(* CoDeSys 2.3.9.59 project: Festo_Project_Group_S.pro *)
(* Title: Tesi *)
(* Version: Studenti *)
(* Author: Marco Pierantoni *)
(* Libraries: STANDARD.LIB 4.10.05 11:14:46, IECSFC.LIB 2.6.14 10:37:46, ANALYZATION.LIB 2.6.14 10:37:46 *)

(* Task configuration *)
TASK SimulationTask (PRIORITY := 1, INTERVAL := T#1ms);
	Pulsantiera();
	PlantCarico();
	PlantScarico();
	PlantMagazzino();
	PlantVerification();
	PlantLavorazione();
	PlantAssemblaggio();
END_TASK
TASK Main (PRIORITY := 1, INTERVAL := T#2ms);
	InputBridge();
	Main();
	OutputBridge();
END_TASK

(* Global variable list: SignalManagement/FaultVariables_List *)
VAR_GLOBAL
(*FAULT VAR*) (* Used as ActivationSignal for SignalManagment *)

	(* Station ONE *)

	F_Cylinder1: BOOL;
	F_S_Cylinder1: BOOL;
	F_A_Cylinder1: BOOL;
	FH_A_Cylinder1: BOOL;
	FL_A_Cylinder1: BOOL;
	FL_DS_Cylinder1: BOOL;
	FH_DS_Cylinder1: BOOL;
	FL_ES_Cylinder1: BOOL;
	FH_ES_Cylinder1: BOOL;

	F_Rotary1: BOOL;
	F_S_Rotary1: BOOL;
	F_A_Rotary1 : BOOL;
	FL_EA_Rotary1: BOOL;
	FH_EA_Rotary1: BOOL;
	FL_DA_Rotary1: BOOL;
	FH_DA_Rotary1: BOOL;
	FL_ES_Rotary1: BOOL;
	FH_ES_Rotary1: BOOL;
	FL_DS_Rotary1: BOOL;
	FH_DS_Rotary1: BOOL;

	F_Vacuum1: BOOL;
	F_S_Vacuum1: BOOL;
	F_A_Vacuum1: BOOL;
	FH_A_Vacuum1: BOOL;
	FL_A_Vacuum1: BOOL;
	FH_S_Vacuum1: BOOL;
	FL_S_Vacuum1: BOOL;

	F_Expulsion1: BOOL;				(* THINK DIAGNOSTIC *)
	F_A_Expulsion1 : BOOL;
	FH_A_Expulsion1: BOOL;
	FL_A_Expulsion1: BOOL;

	(* Station TWO *)

	F_Elevator2: BOOL;
	F_S_Elevator2: BOOL;
	F_A_Elevator2: BOOL;
	FH_EA_Elevator2: BOOL;
	FL_EA_Elevator2: BOOL;
	FH_DA_Elevator2: BOOL;
	FL_DA_Elevator2: BOOL;
	FH_ES_Elevator2: BOOL;
	FL_ES_Elevator2: BOOL;
	FH_DS_Elevator2: BOOL;
	FL_DS_Elevator2: BOOL;

	F_Cylinder2: BOOL;
	F_S_Cylinder2: BOOL;
	F_A_Cylinder2: BOOL;
	FH_A_Cylinder2 : BOOL;
	FL_A_Cylinder2 : BOOL;
	FH_S_Cylinder2 : BOOL;
	FL_S_Cylinder2 : BOOL;

	F_Air2: BOOL;				(* THINK DIAGNOSTIC *)
	F_S_Air2: BOOL;
	F_A_Air2: BOOL;
	FH_A_Air2: BOOL;
	FL_A_Air2: BOOL;

	(* Station THREE *)

	F_RotaryTable3: BOOL;
	F_S_RotaryTable3: BOOL;
	F_A_RotaryTable3: BOOL;
	FH_A_RotaryTable3: BOOL;
	FL_A_RotaryTable3: BOOL;
	FH_S_RotaryTable3: BOOL;
	FL_S_RotaryTable3: BOOL;

	F_Cylinder3: BOOL;		(* THINK DIAGNOSTIC *)
	F_S_Cylinder3: BOOL;
	F_A_Cylinder3: BOOL;
	FH_A_Cylinder3: BOOL;
	FL_A_Cylinder3: BOOL;

	F_DrillCylinder3: BOOL;
	F_S_DrillCylinder3: BOOL;
	F_A_DrillCylinder3: BOOL;
	FH_EA_DrillCylinder3: BOOL;
	FL_EA_DrillCylinder3: BOOL;
	FH_DA_DrillCylinder3: BOOL;
	FL_DA_DrillCylinder3: BOOL;
	FH_ES_DrillCylinder3: BOOL;
	FL_ES_DrillCylinder3: BOOL;
	FH_DS_DrillCylinder3: BOOL;
	FL_DS_DrillCylinder3: BOOL;

	F_Drilling3: BOOL;			(* THINK DIAGNOSTIC *)
	F_S_Drilling3: BOOL;
	F_A_Drilling3: BOOL;
	FH_A_Drilling3: BOOL;
	FL_A_Drilling3: BOOL;

	F_Block3: BOOL;			(* THINK DIAGNOSTIC *)
	F_S_Block3: BOOL;
	F_A_Block3: BOOL;
	FH_A_Block3: BOOL;
	FL_A_Block3: BOOL;

	F_Expell3: BOOL;				(* THINK DIAGNOSTIC *)
	F_S_Expell3: BOOL;
	F_A_Expell3: BOOL;
	FH_A_Expell3: BOOL;
	FL_A_Expell3: BOOL;

	(* Station FOUR *)

	F_SpringExtractor4: BOOL;
	F_S_SpringExtractor4: BOOL;
	F_A_SpringExtractor4: BOOL;
	FH_A_SpringExtractor4: BOOL;
	FL_A_SpringExtractor4: BOOL;
	FH_ES_SpringExtractor4: BOOL;
	FL_ES_SpringExtractor4: BOOL;
	FH_DS_SpringExtractor4: BOOL;
	FL_DS_SpringExtractor4: BOOL;

	F_PistonSelector4: BOOL;
	F_S_PistonSelector4: BOOL;
	F_A_PistonSelector4: BOOL;
	FH_EA_PistonSelector4: BOOL;
	FL_EA_PistonSelector4: BOOL;
	FH_DA_PistonSelector4: BOOL;
	FL_DA_PistonSelector4: BOOL;
	FH_ES_PistonSelector4: BOOL;
	FL_ES_PistonSelector4: BOOL;
	FH_DS_PistonSelector4: BOOL;
	FL_DS_PistonSelector4: BOOL;

	F_ExtractCover4: BOOL;
	F_S_ExtractCover4: BOOL;
	F_A_ExtractCover4: BOOL;
	FH_A_ExtractCover4: BOOL;
	FL_A_ExtractCover4: BOOL;
	FH_ES_ExtractCover4: BOOL;
	FL_ES_ExtractCover4: BOOL;
	FH_DS_ExtractCover4: BOOL;
	FL_DS_ExtractCover4: BOOL;

	F_BlockingCylinder4: BOOL;		(* THINK DIAGNOSTIC *)
	F_S_BlockingCylinder4: BOOL;
	F_A_BlockingCylinder4: BOOL;
	FH_A_BlockingCylinder4: BOOL;
	FL_A_BlockingCylinder4: BOOL;

	(* Robot Manipulator *)

	F_A_RobotToInitial4: BOOL;
	F_S_RobotInInitial4: BOOL;
	(*F_A_RobotTakeBlack4: BOOL;
	F_A_RobotTakeRedSilver4: BOOL;
	F_A_RobotDiscardBlack4: BOOL;
	F_A_RobotDiscardRedSilver4: BOOL;*)
	F_A_RobotAssembly4: BOOL;
	F_S_RobotAssembly4: BOOL;
	F_A_RobotPiston4: BOOL;
	F_S_RobotPiston4: BOOL;
	F_A_RobotSpring4: BOOL;
	F_S_RobotSpring4: BOOL;
	F_A_RobotCover4: BOOL;
	F_S_RobotCover4: BOOL;
	(*F_A_RobotReset4: BOOL;*)

END_VAR

(* Global variable list: MyGlobal/GenericDeviceLib *)
(*Feedback*)

VAR_GLOBAL CONSTANT
	DEVICE_WITHOUT_FEEDBACK : BYTE := 2#01000000;
	DEVICE_WITH_ENABLE_FEEDBACK : BYTE := 2#00010000;
	DEVICE_WITH_DISABLE_FEEDBACK : BYTE := 2#00100000;
	DEVICE_WITH_DOUBLE_FEEDBACK : BYTE := 2#00110000;
	DEVICE_FEEDBACK_MASK : BYTE := 2#11110000;
END_VAR

(*Actuation*)

VAR_GLOBAL CONSTANT
	DEVICE_WITH_SINGLE_ACTUATION : BYTE := 2#00000001;
	DEVICE_WITH_DOUBLE_ACTUATION : BYTE := 2#00000011;
	DEVICE_WITH_DA_NO_RETAIN : BYTE := 2#00000010;
	DEVICE_ACTUATION_MASK : BYTE := 2#00001111;
END_VAR

(* Global variable list: MyGlobal/My_global *)
VAR_GLOBAL CONSTANT

	INIT : INT := 1;
	RUN : INT := 2;
	IMMEDIATESTOPMACHINE : INT :=3;
	READYTORESET : INT:= 4;
	READYTORUN : INT := 5;
	ONPHASESTOPMACHINE : INT := 6;
	EMERGENCYSTOPMACHINE : INT := 7;

END_VAR

VAR_GLOBAL

	BridgeInitOperation : BOOL := TRUE; (* USED ONLY for RealPlant *)
	SignHandlerOperationType : INT ;
	DeviceClock : BOOL;
	OperationType : INT;
	KeyReset : BOOL;
	CumulativeReset : BOOL;
	NoSignalsToReset : BOOL;
	OUTPUT_COUNTER_DELAY : INT := 5; (* Used for Provisional Reset , equal for all by design*)
	SensorActuationDiagnosticEnabled : BOOL := TRUE;

	AllStationsIdle: BOOL; (*Needed For Auto-Stop in case of Inactivity*)

	EmergencyInStop : BOOL;
	ImmediateInStop : BOOL;
	OnPhaseInStop : BOOL;

	(* Necessary on Virtual Panel *)

	VL_StateInit: BOOL;
	VL_StateReady: BOOL;
	VL_StateRun: BOOL;
	VL_StateAlarm: BOOL;
	VL_StateImmediateStop: BOOL;
	VL_StateStop: BOOL;
	VL_StateReset: BOOL;

	VL_ColorVis2:DWORD;
	VL_ColorVis3:DWORD;
	VL_ColorVis:DWORD;
	VL_PositionVis: DWORD;
	VL_ColorVis4:DWORD;
	VL_Completed: INT;
	VL_Rejected: INT;

	(* Used for Station 4 *)

	SpringHouseNotEmpty: BOOL;
	B_SpringLoader: BOOL;
	NumSpring: INT := 0;
	B_PistonLoader: BOOL;
	PistonHouseNotEmpty: BOOL;
	NumPistonBlack: INT;
	NumPistonGrey: INT;

	(*Needed global for real plant for filters*)
	(*Clock2ms: BOOL;
	Clock10ms: BOOL;
	Clock100ms: BOOL;
	Clock1s: BOOL;*)

END_VAR

(* Global variable list: MyGlobal/MyBridgedVariables *)
VAR_GLOBAL

(******* My Variables for Sensors (S), Actuators (A), Lights (L) and Buttons (B)  ***************)

	(* Distribution Station *)

	S_EmptyWarehouse1: BOOL;
	S_CylinderExtended1:BOOL;
	A_Cylinder1: BOOL;
	S_CylinderRetracted1: BOOL;
	A_ArmToWarehouse1: BOOL;
	A_ArmToElevator1: BOOL;
	S_ArmInWarehouse1: BOOL;
	S_ArmInElevator1: BOOL;
	A_Vacuum1: BOOL;
	S_VacuumOk1: BOOL;
	A_AirVacuum1: BOOL;

	(* Verification/Testing Station *)

	S_InterferenceArmElevator2: BOOL;
	A_ElevatorUp2: BOOL;
	A_ElevatorDown2: BOOL;
	S_IsElevatorUp2: BOOL;
	S_IsElevatorDown2: BOOL;
	A_Cylinder2: BOOL;
	S_CylinderExtended2: BOOL;
	S_CylinderRetracted2: BOOL;
	A_AirSlider2: BOOL;
	S_ElementInElevator2: BOOL;
	S_Color2: BOOL;
	S_IsHigh2: BOOL;

	(* Processing Station *)

	A_RotaryTable3: BOOL;
	S_RotaryAlligned3: BOOL;
	S_AvaiableElement3: BOOL;
	S_ControlElement3: BOOL;
	S_DrillElement3: BOOL;
	A_GoControl3: BOOL;
	S_IsOnTheRightSide3: BOOL;
	A_GoDrill3: BOOL;
	A_ReturnDrill3: BOOL;
	S_DrillUp3: BOOL;
	S_DrillDown3: BOOL;
	A_Drilling3: BOOL;
	A_BlockElement3: BOOL;
	A_ExpellElement3: BOOL;

	(* Assembly Station *)

	A_SpringCylinder4: BOOL;
	S_SpringCylinderExtended4: BOOL;
	S_SpringCylinderRetracted4: BOOL;
	A_GiveBlackPiston4: BOOL;
	A_GiveSilverPiston4: BOOL;
	S_BlackPistonGiven4: BOOL;
	S_SilverPistonGiven4: BOOL;
	A_CoverCylinder4: BOOL;
	S_NoCover4: BOOL;
	S_CoverCylinderRetracted4: BOOL;
	S_CoverCylinderExtracted4: BOOL;
	S_ElementAvailable4: BOOL;
	A_BlockElement4: BOOL;

	(* Robot Manipulator *)

	A_RobotToInitial4: BOOL;
	S_RobotInInitial4: BOOL;
	A_RobotTakeBlack4: BOOL;
	A_RobotTakeRedSilver4: BOOL;
	A_RobotDiscardBlack4: BOOL;
	 A_RobotDiscardRedSilver4: BOOL;
	A_RobotAssembly4: BOOL;
	S_RobotAssembly4: BOOL;
	A_RobotPiston4: BOOL;
	S_RobotPiston4: BOOL;
	A_RobotSpring4: BOOL;
	S_RobotSpring4: BOOL;
	A_RobotCover4: BOOL;
	S_RobotCover4: BOOL;
	A_RobotReset4: BOOL;
	StopOutput4 : BOOL := FALSE;

	(* Buttons and Lights *)

	B_Start: BOOL;
	L_Start: BOOL;
	B_Reset: BOOL;
	L_Reset: BOOL;
	B_Stop: BOOL;
	B_Freeze: BOOL;
	B_Emergency: BOOL;
	L_PieceToDiscard2 : BOOL;
	L_EmptyWarehouse: BOOL;
	B_FullWarehouse: BOOL;
	L_UpsideDownElement: BOOL;
	L_NoCover: BOOL;
	B_OnlyBlackElement: BOOL;
	B_AllColors: BOOL;
	B_FaultyElementRemoved: BOOL;
	L_RobotMoving: BOOL;
	L_RobotOn: BOOL;
	L_BlackElement: BOOL;
	L_RedSilverElement: BOOL;
	B_FillAll:BOOL;

END_VAR

(* Global variable list: SignalManagement/SignalCodes_List *)
VAR_GLOBAL

	(*FAULT MESSAGE*) (* "SignalCodes" *)

	(* ALARMS : 1-70 *)

	(*ANOMALIES : 71-130 *)

	(* Warnings: 131 - 190 *)

	(* Informations : 191 - 256 *)

(************************************************************************************************************************************)

	(* Each type has first 10 for Others, 10 for S1, 10 for S2, 10 for S3, 10 for S4 and 10 or more for Others *)

	(*PRIORITARY ALARMS *)

	mEmergencyButtonPressed : WORD := 0003;
	mFreezeButtonPressed : WORD := 0004;
	mOnPhaseStopButtonPressed : WORD := 0005;

	(* WARNINGS *)

	mIdleStopAutoRequest : WORD := 00131;

	(* INFORMATIONS *)

	mEmptyWarehouse : WORD := 00191;
	mEmpyCoverInAssembly : WORD := 00198;

	(*DISTRIBUTION STATION *)

	mS1CylinderActuationFault : WORD := 00021;				mS1CylinderSensorFault : WORD := 00081;
	mS1ArmActuationFault : WORD := 00023;					mS1ArmSensorFault : WORD := 00084;
	mS1VacuumActuationFault : WORD := 00026; 				mS1VacuumSensorFault : WORD := 00087;
	mS1ExpulsionAirActuationFault : WORD := 00028;

	(*VERIFICATION STATION *)

	mS2ElevatorActuationFault : WORD := 00031; 		 		mS2ElevatorSensorFault : WORD := 00091;
	mS2CylinderActuationFault : WORD := 00034; 		 		mS2CylinderSensorFault : WORD := 00094;
	mS2AirSliderActuationFault : WORD := 00036;
	
	(*PROCESSING STATION *)

	mS3RotaryActuationFault : WORD := 00041;	 		  		mS3RotarySensorFault : WORD := 00101;
	mS3InspectorActuationFault : WORD := 00043;	
	mS3DrillCylinderActuationFault : WORD := 00045; 	  		mS3DrillCylinderSensorFault : WORD := 00103;
	mS3DrilerActuationFault : WORD := 00047;
	mS3BlockerActuationFault : WORD := 00048;
	mS3ExpellerActuationFault : WORD := 00049;

	(*ASSEMBLY STATION *)

	mS4SpringExtractorActuationFault : WORD := 00051;		mS4SpringExtractorSensorFault : WORD := 00111;
	mS4PistonSelectorActuationFault : WORD := 00052;		mS4PistonSelectorSensorFault : WORD := 00112;
	mS4CoverExtractorActuationFault : WORD := 00053;		mS4CoverExtractorSensorFault: WORD := 00113;
	mS4BlockerActuationFault : WORD := 00054;

	(* ROBOT MANIPULATOR *)

	mS4RobotInitActuationFault : WORD := 00056;				mS4RobotInitSensorFault : WORD := 00115;
	mS4RobotPistonActuationFault : WORD := 00057;			mS4RobotPistonSensorFault : WORD := 00116;
	mS4RobotSpringActuationFault : WORD := 00058;			mS4RobotSpringSensorFault : WORD := 00117;
	mS4RobotCoverActuationFault : WORD := 00059;			mS4RobotCoverSensorFault : WORD := 00118;
	mS4RobotAssemblyActuationFault : WORD := 00060;		mS4RobotAssemblySensorFault : WORD := 00119;

END_VAR

(* Global variable list: SignalManagement/SignalConstants *)
VAR_GLOBAL CONSTANT
(* OperationTypes *)

(*	INIT : INT :=1;	*)

	START_CONFIGURATION : INT := 12;
	CONFIGURATION : INT := 13;
	START_GENERATION : INT := 14;
	GENERATION : INT := 15;

(* SignalTypes *)

	ALARM : WORD := 00001;
	ANOMALY : WORD := 00002;
	WARNING : WORD := 00003;
	INFORMATION : WORD := 00004;
	SIGNAL_TYPE_MASK : WORD := 00007;

(* ResetTypes *)

	AUX_RESET : WORD := 512;			 (* Reset enabled only if aux reset input active *)
	AUTO_RESET : WORD := 1024;		(* IF ActivationSignal is not present anymore *)
	AUTO_CONDITIONED_RESET : WORD := 2048;	(* IF ActivatSignal not pres anymore AND IF AutoResetSignal TRUE *)
	UNCONDITIONED_RESET : WORD := 4096;		(* Reset in any case if most important *)

	AUTO_PROVISIONAL_RESET : WORD := 8192;
	AUTO_PRIORITY_RESET : WORD := 16384;

(* SignalOutputs *)

	NONE : DWORD := 16#000;

	EMERGENCY_STOP : DWORD := 16#0001;
	IMMEDIATE_STOP : DWORD := 16#0002;
	ON_PHASE_STOP : DWORD := 16#0004;

END_VAR

(* Global variable list: SIM_Global_Variables *)
VAR_GLOBAL


(*------------------------------------------------------------------------------------------------------------------------------------------------*)
(*-----------------------------------VARIABILI DI VISUALIZZAZIONE DEGLI ELEMENTI----------------------------------------*)

(********************variabili utilizzate solo per la simulazione (NON per la logica di controllo)**********************)

(*---------Elementi presenti nel magazzino basi: il magazzino può contenere al più 8 elementi---------*)
	ElementOneCharged: BOOL; (*variabile che indica la presenza del primo elemento nel magazzino*)
	ElementTwoCharged: BOOL; (*secondo elemento caricato nel magazzino*)
	ElementThreeCharged: BOOL; (*terzo elemento caricato nel magazzino*)
	ElementFourCharged: BOOL; (*quarto elemento caricato nel magazzino*)
	ElementFiveCharged: BOOL; (*quinto elemento caricato nel magazzino*)
	ElementSixCharged: BOOL; (*sesto elemento caricato nel magazzino*)
	ElementSevenCharged: BOOL; (*settimo elemento caricato nel magazzino*)
	ElementEightCharged: BOOL; (*ottavo e ultimo elemento caricato nel magazzino*)

(*colori. I possibili colori degli elementi caricabili sono: Rosso, Nero e Argentato (o Metallico)*)
	Red: BOOL; (*è stato caricato un pezzo rosso*)
	Black: BOOL; (*è stato caricato un pezzo nero*)
	Silver: BOOL; (*è stato caricato un pezzo argentato*)

(*pezzi rossi*)
	ElementOneRed: BOOL; (*variabile che indica che il primo elemento caricato è rosso*)
	ElementTwoRed: BOOL; (*il secondo elemento caricato è rosso*)
	ElementThreeRed: BOOL; (*il terzo elemento caricato è rosso*)
	ElementFourRed: BOOL; (*il quarto elemento caricato è rosso*)
	ElementFiveRed: BOOL; (*il quinto elemento caricato è rosso*)
	ElementSixRed: BOOL; (*il sesto elemento caricato è rosso*)
	ElementSevenRed: BOOL; (*il settimo elemento caricato è rosso*)
	ElementEightRed: BOOL; (*l'ottavo elemento caricato è rosso*)

 (*pezzi metallici*)
	ElementOneSilver: BOOL; (*variabile che indica che il primo elemento caricato è argentato*)
	ElementTwoSilver: BOOL;
	ElementThreeSilver: BOOL;
	ElementFourSilver: BOOL;
	ElementFiveSilver: BOOL;
	ElementSixSilver: BOOL;
	ElementSevenSilver: BOOL;
	ElementEightSilver: BOOL;

 (*pezzi neri*)
	ElementOneBlack: BOOL; (*variabile che indica che il primo elemento caricato è nero*)
	ElementTwoBlack: BOOL;
	ElementThreeBlack: BOOL;
	ElementFourBlack: BOOL;
	ElementFiveBlack: BOOL;
	ElementSixBlack: BOOL;
	ElementSevenBlack: BOOL;
	ElementEightBlack: BOOL;

(*-----pezzi capovolti-----Può capitare che alcune basi vengano caricate capovolte nel magazzino: le variabili seguenti simulano questa ipotesi*)
	Redoverturned: BOOL; (*variabile che indica che l'elemento rosso è capovolto*)
	Silveroverturned: BOOL; (*variabile che indica che l'elemento argentato è capovolto*)
	Blackoverturned: BOOL; (*variabile che indica che l'elemento nero è capovolto*)

(*---------Elementi caricati capovolti nel magazzino basi--------*)
	ElementOneOverturned: BOOL; (*variabile che indica che il primo elemento del magazzino è stato caricato capovolto*)
	ElementTwoOverturned: BOOL; (*secondo elemento del magazzino caricato capovolto*)
	ElementThreeOverturned: BOOL; (*terzo elemento del magazzino caricato capovolto*)
	ElementFourOverturned: BOOL; (*quarto elemento del magazzino caricato capovolto*)
	ElementFiveOverturned: BOOL; (*quinto elemento del magazzino caricato capovolto*)
	ElementSixOverturned: BOOL; (*sesto elemento del magazzino caricato capovolto*)
	ElementSevenOverturned: BOOL; (*settimo elemento del magazzino caricato capovolto*)
	ElementEightOverturned: BOOL; (*ottavo elemento del magazzino caricato capovolto*)

(*----pezzi corti:
I pezzi chiari (rossi/met) sono alti, quelli neri, bassi. Può capitare che nel magazzino vengano caricati pezzi chiari ma bassi per difetti di costruzione:
le variabili seguenti simulano questa ipotesi*)

(*per la simulazione è stato creato solo il pezzo metallico corto: non è necessario creare anche quello rosso perchè il sistema non distingue tra rosso e metallico ma solo tra chiaro e nero*)
	Silvershort: BOOL; (*pezzo argentato corto*)

(*---------Elementi corti caricati nel magazzino basi--------*)
	ElementOneShort: BOOL; (*il primo elemento del magazzino è corto*)
	ElementTwoShort: BOOL;
	ElementThreeShort: BOOL;
	ElementFourShort: BOOL;
	ElementFiveShort: BOOL;
	ElementSixShort: BOOL;
	ElementSevenShort: BOOL;
	ElementEightShort: BOOL;

(*stringhe di segnalazione pezzo capovolto o corto: viene visualizzata una O se il pezzo è capovolto oppure una S se è corto. Niente altrimenti.*)
	ElementOneO: STRING; (*sul primo elemento del magazzino viene visualizzata stringa "O"(Overturned), oppure "S" (Short), oppure "" (pezzo normale)*)
	ElementTwoO: STRING;
	ElementThreeO: STRING;
	ElementFourO: STRING;
	ElementFiveO: STRING;
	ElementSixO: STRING;
	ElementSevenO: STRING;
	ElementEightO: STRING;

(*-----Elemento in Attesa: una volta espulso dal magazzino basi l'elemento rimane in attesa di essere caricato dal braccio rotante-----*)
	ElementWaitingCharged: BOOL; (*variabile che indica che è presente un elemento in attesa*)
	ElementWaitingRed: BOOL; (*variabile che indica che l'elemento in attesa è rosso*)
	ElementWaitingBlack: BOOL; (*variabile che indica che l'elemento in attesa è nero*)
	ElementWaitingSilver: BOOL; (*variabile che indica che l'elemento in attesa è argentato*)
	ElementWaitingOverturned: BOOL; (*variabile che indica che l'elemento in attesa è capovolto*)
	ElementWaitingShort: BOOL; (*variabile che indica che l'elemento in attesa è corto*)
	ElementWaitingO: STRING; (*stringa di segnalazione elemento in attesa capovolto o corto*)

(*------------Elemento sul Braccio rotante-------------*)
	ElementRotaryCharged: BOOL; (*variabile che indica che un elemento è caricato sul braccio rotante*)
	ElementRotaryRed: BOOL;
	ElementRotaryBlack: BOOL;
	ElementRotarySilver: BOOL;
	ElementRotaryOverturned: BOOL;
	ElementRotaryShort: BOOL;
	ElementRotaryO: STRING;

(*------------------Elemento in Verifica--------------------*)
	ElementVerificationCharged: BOOL;  (*variabile che indica che è presente un elemento nella stazione di verifica*)
	ElementVerificationRed: BOOL;
	ElementVerificationBlack: BOOL;
	ElementVerificationSilver: BOOL;
	ElementVerificationOverturned: BOOL;
	ElementVerificationShort: BOOL;
	ElementVerificationO: STRING;

(*------------------Elemento Misura----------------------*)
	ElementMeasureCharged: BOOL; (*variabile che indica che un elemento è giunto sotto al misuratore*)
	ElementMeasureRed: BOOL;
	ElementMeasureSilver: BOOL;
	ElementMeasureBlack: BOOL;
	ElementMeasureOverturned: BOOL;
	ElementMeasureShort: BOOL;
	ElementMeasureO: STRING;

(*--------------Elemento Cuscinetto d'aria--------------*)
	ElementAirCharged: BOOL;  (*variabile che indica la presenza di un elemento sulla guida a cuscinetto d'aria*)
	ElementAirRed: BOOL;
	ElementAirSilver: BOOL;
	ElementAirBlack: BOOL;
	ElementAirOverturned: BOOL;
	ElementAirO: STRING;



																			(*ATTUATORI E SENSORI*)
(*xxxxxxxxxxxxxxxxxxxxxxxxxxxxxxxxxxxxxxxxxxxxxxxxxxxxxxxxxxxxxxxxxxxxxxxxxxxxxxxxxxxxxxxxxxxxxxxxxxxxxxxxxxxxxxxxxxxxxxxxxxxxxxxxxxxxxxxxxxxxxxxxxxxxxxxxxxxxxxxxxxxxxxxxxxxxxxxxxxxxxxxxxxxxxxxxxx*)

(* -------------MODULO MAGAZZINO DI STOCCAGGIO (magazzino basi) -----------*)

(*variabili associate ad attuatori e sensori: (***utilizzate nella logica di controllo***)*)
	EmptyWarehouse:BOOL;  (*sensore magazzino pezzi vuoto*)
	CylinderExtractionLoadInExtensivePosition:BOOL; (*sensore cilindro di estrazione in posizione estratta*)
	CylinderExtractionLoadInRetroactivePosition:BOOL; (*sensore cilindro di estrazione in posizione retratta*)
	CylinderExtractsLoadFromWarehouse:BOOL; (*comando di estrazione pezzo dal magazzino *)

(*variabili della simulazione *)
	CylinderPosition: INT; (* variabile utilizzata per simulare il movimento del cilindro di estrazione *)
	ElementPosition: INT; (* variabile utilizzata per simulare il movimento dell'elemento in uscita dal magazzino *)
	CylinderBehind:BOOL; (*variabile che indica che il cilindro sta tornando indietro *)

(*----------------- MODULO DI TRASFERIMENTO (braccio rotante) ---------------*)

(*variabili associate ad attuatori e sensori: (***utilizzate nella logica di controllo***)*)
	RotaryMakerVsWarehouse:BOOL;  (*comando rotary maker verso magazzino pezzi *)
	RotaryMakerVsVerification:BOOL;  (*comando rotary maker verso stazione di verifica *)
	RotaryMakerInPositionWarehouse:BOOL;  (*sensore di finecorsa rotary maker in posizione magazzino pezzi *)
	RotaryMakerInPositionVerification:BOOL;  (*sensore di finecorsa rotary maker in stazione di verifica *)
	VacuumGenerator:BOOL;  (*comando generatore di vuoto *)
	VacuumGeneratorOk:BOOL;  (*sensore di vuoto*)
	ExpulsionAirVacuum:BOOL;  (*comando getto d'aria per espulsione *)

(*variabili della simulazione *)
	RotaryPosition: INT; (* variabile utilizzata per simulare il movimento del rotary maker *)
       ReadyForRotaryMaker: BOOL; (* variabile di simulazione che indica la disponibilità di un pezzo per il braccio rotante*)
	VacuumGeneratorSim: BOOL; (*simulazione generatore di vuoto*)
	ExpulsionAirVacuumVis:BOOL; (*visualizzazione getto d'aria per espulsione *)

(*simulazione valore iniziale braccio rotante: *)
	RotaryPositionInitialVis: INT; (*variabile intera che indica la posizione in cui si trova il braccio rotante prima della simulazione*)
	FLAGRotaryPosition: BOOL := TRUE;

(* -------------------------------------STAZIONE DI VERIFICA------------------------------- *)

(*variabili associate ad attuatori e sensori: (***utilizzate nella logica di controllo***)*)
	VerificationBusy: BOOL; (*sensore a fotocellula per interferenza braccio rotante-ascensore*)
	ToLiftCylinderToMeasureLoad:BOOL; (*comando modulo di sollevamento verso l'alto *)
	ToLowerCylinderToMeasureLoad:BOOL; (*comando modulo di sollevamento verso il basso *)
	CylinderUpToMeasureLoad:BOOL;  (*sensore finecorsa modulo di sollevamento in alto *)
	CylinderDownToMeasureLoad:BOOL; (*sensore finecorsa modulo di sollevamento in basso *)
	ToExtendCylinderOfExtractionVsGuide:BOOL; (*comando espulsione pezzo *)
	CylinderOfExtractionInRetroactivePosition:BOOL; (*sensore finecorsa cilindro di estrazione in posizione retratta *)
       CylinderOfExtractionInExtensivePosition:BOOL; (*sensore finecorsa cilindro di estrazione in posizione estesa (Virtuale) *)
       ResetVirtualSensorElevator: BOOL; (*Serve a resettare il sensore virtuale dell'elevatore a seguito di un plausibile Fault*)

       AirCushion:BOOL; (*comando cuscinetto d'aria*)
	ReadyLoadForVerification:BOOL; (*sensore presenza pezzo alla base della stazione di verifica *)
	ColourMeasurement:BOOL; (*sensore di rilevazione colore: 0 nero, 1 rosso/metallico *)
	MeasurementNotOk: BOOL; (*sensore di misuarazione altezza. Uscita del misuratore: 1 pezzo alto, 0 pezzo basso*)

(*variabili della simulazione *)
	LiftPosition: INT; (* variabile utilizzata per simulare il movimento del modulo di sollevamento *)
	CylinderOfExtractionPosition:INT; (* variabile utilizzata per simulare il movimento del cilindro espulsione *)
	MisuratorPosition: INT; (* variabile utilizzata per simulare il movimento del misuratore*)
	MovementElementAir: INT; (* variabile utilizzata per simulare il movimento dell'elemento sul cuscino d'aria*)
	AirCushionVis: BOOL; (*visualizzazione cuscinetto d'aria*)
	ElementAirVsRotaryTable: BOOL; (*variabile di simulazione che notifica l'arrivo dell'elemento d'aria sulla tavola rotante*)

(*simulazione valore iniziale modulo di sollevamento*)
	LiftPositionInitialVis: INT;  (*variabile intera che indica la posizione in cui si trova l'ascensore prima della simulazione*)
	FLAGLiftPosition: BOOL:=TRUE;

(*STAZIONE DI LAVORAZIONE*)

	(* MODULO TAVOLA ROTANTE*)
	RotaryTableMotor:BOOL; (* COMANDO DI ATTUAZIONE: tavola rotante *)
	AlignementRotaryTableWithPositionings:BOOL; (* SENSORE: tavola allineata con le postazioni *)
       AvailableLoadForWorkingStation:BOOL; (* SENSORE DI PRESENZA: load presente nella prima stazione della giostra*)
       AvailableLoadInControlPositioning:BOOL; (*SENSORE DI PRESENZA: load presente in postazione di controllo*)
       AvailableLoadInDrillingPositioning:BOOL; (*SENSORE DI PRESENZA: load presente nel modulo di foratura*)

	(* MODULO DI CONTROLLO*)
	ToLowerCylinderToInspectLoad:BOOL; (* COMANDO DI ATTUAZIONE: L'unità di controllo viene abbassata *)
	InControlLoadInWrongPositionToBeDrilled: BOOL; (*SENSORE per il rilevamento del corretto orientamento della base*)

      	(* MODULO DI FORATURA.*)
	ToLiftDrillingUnit:BOOL; (*COMANDO DI ATTUAZIONE:  l'unità di foratura viene abbassata *)
	ToLowerDrillingUnit:BOOL; (*COMANDO DI ATTUAZIONE: l'unità di foratura viene sollevata *)
	DrillingUnitUp:BOOL; (* SENSORE: unità di foratura in posizione sollevata*)
	DrillingUnitDown:BOOL; (* SENSORE: unità di foratura sulla base del pezzo *)
	DrillingUnitActive:BOOL; (* COMANDO DI ATTUAZIONE: unità di foratura ruota in senso orario *)
	BlockingCylinderForwardInDrillingPositioning:BOOL; (*COMANDO DI ATTUAZIONE: pistone di bloccaggio pezzo*)
       DrillingUnitClockWise:BOOL;
       (* MODULO DI ESPULSIONE.*)
       ExpellingLeverActive:BOOL; (*COMANDO DI ATTUAZIONE:  leva espelle pezzo *)


	(*STAZIONE DI ASSEMBLAGGIO*)

 	(* MODULO MOLLE.*)
	ToExtractSpringInAssemblyStation:BOOL; (* COMANDO DI ATTUAZIONE del cilindro che preleva la molla dal magazzino *)
	ToExtractSpringInAssemblyStationInExtensivePosition:BOOL; (* SENSORE di fine corsa che indica che il cilindro è in posizione estesa(di riposo)*)
	ToExtractSpringInAssemblyStationInRetroactivePosition:BOOL; (*SENSORE di fine corsa che indica che il cilindro è in posizione ritratta*)

	(* MODULO MAGAZZINO  PISTONI.*)
	PistonSelectorGoOnTheRight:BOOL; (*COMANDO DI ATTUAZIONE: magazzino pistoni ruota verso destra (preleva pistone NERO)*)
	PistonSelectorGoOnTheLeft:BOOL; (*COMANDO DI ATTUAZIONE: magazzino pistoni ruota verso sinistra(preleva pistone GRIGIO)*)
	PistonSelectorIsOnTheRight:BOOL; (* SENSORE: magazzino pistoni ruotato completamente a destra *)
	PistonSelectorIsOnTheLeft:BOOL; (* SENSORE: magazzino pistoni ruotato completamente a sinistra *)

	(* MODULO STOCCAGGIO COPERCHI.*)
	ToExtractCoverInAssemblyStationForward:BOOL; (*COMANDO DI ATTUAZIONE: cilindro estrae cover *)
	EmptyCoverHouseInAssemblyStation: BOOL; (*SENSORE: segnala se sono presenti dei coperchi nel magazzino*)
	ToExtractCoverInAssemblyStationInRetroactivePosition:BOOL; (*SENSORE:  cilindro di estrazione in posizione retratta *)
	ToExtractCoverInAssemblyStationInExtensivePosition:BOOL; (*SENSORE: cilindro di estrazione in posizione estesa *)

	(*STAZIONE1 DOPO LA GIOSTRA*)
	AvailableLoadForRobot:BOOL; (*SENSORE: nella stazione1 dopo la giostra, indica la presenza di una base pronta per l'assemblaggio*)
	(*STAZIONE DI ASSEMBLAGGIO PEZZO*)
	BlockingCylinderForwardInAssemblyStation:BOOL;  (*COMANDO DI ATTUAZIONE: cilindro di boccaggio, SE TRUE SI SBLOCCA il pezzo *)
	(*POSIZIONE INIZIALE ROBOT*)
	RobotGoToInitialPosition: BOOL; (*COMANDO DI ATTUAZIONE: porta il robot nella posizione iniziale*)
	RobotInInitialPosition: BOOL; (*SENSORE: indica che il robot è arrivato nella posizione iniziale*)

	(*STAZIONE DI ASSEMBLAGGIO*)
	RobotTakeBlackLoad: BOOL; (*COMANDO DI ATTUAZIONE : impone al robot la sequenza di istruzioni tale da prelevare una base Nera*)
	RobotTakeRedSilverLoad: BOOL; (*COMANDO DI ATTUAZIONE : impone al robot la sequenza di istruzioni tale da prelevare una base Rossa-Argento*)
	RobotTakeLoadToDiascardBlack: BOOL; (*COMANDO DI ATTUAZIONE : impone al robot la sequenza di istruzioni tale da prelevare una base Capovolta*)
	RobotTakeLoadToDiascardRedSilver: BOOL; (*COMANDO DI ATTUAZIONE : impone al robot la sequenza di istruzioni tale da prelevare una base Capovolta*)
	RobotTakeCurrentLoadToAssembly: BOOL; (*COMANDO DI ATTUAZIONE : impone al robot la sequenza di istruzioni tale da portare il robot nella stazione di assemblaggio*)

	RobotInAssemblyUnit: BOOL; (*SENSORE: robot in posizione di assemblaggio*)
	(*STAZIONE DEI PISTONI*)
	RobotGoToPistonHouse: BOOL;  (*COMANDO DI ATTUAZIONE: porta il robot nella stazione dei pistoni*)
	RobotInPistonWarehouse: BOOL;  (*SENSORE: robot nella stazione dei pistoni*)
	(*STAZIONE DELLE MOLLE*)
	RobotGoToSpringHouse: BOOL; (*COMANDO DI ATTUAZIONE: porta il robot nella stazione delle molle*)
	RobotInSpringWarehouse:BOOL:=FALSE; (* SENSORE: robot nella stazione delle molle *)
	(*STAZIONE DEI COPERCHI*)
	RobotGoToCoverHouse: BOOL; (*COMANDO DI ATTUAZIONE: porta il robot nella stazione dei coperchi*)
	RobotInCoverWarehouse:BOOL;  (*SENSORE: robot nella stazione dei coperchi*)

	RobotReset:BOOL; (*Inizializzazione del robot da fare alla fine della lavorazione di un pezzo*)

	(*VARIABILI DI CONTROLLO utilizzate anche nella simulazione*)
	Fault: BOOL; (*Variabile di visualizzazione: se true rende visibile il display "Fault" *)
	FaultDetected: BOOL; (*GUASTO RILEVATO, per far ripartire il sistema dopo un fault che non necessita di riavvio*)
	EmergencyRobot: BOOL; (*Variabile per fermare il robot in caso di emergenza*)
(*xxxxxxxxxxxxxxxxxxxxxxxxxxxxxxxxxxxxxxxxxxxxxxxxxxxxxxxxxxxxxxxxxxxxxxxxxxxxxxxxxxxxxxxxxxxxxxxxxxxxxxxxxxxxxxxxxxxxxxxxxxxxxxxxxxxxxxxxxxxxxxxxxxxxxxxxxxxxxxxxxxxxxxxxxxxxxxxxxxxxxxxxxxxxxxxxxx*)


(*------------------------------------------------------------------------------------------------------------------------------------------------------------------------*)
(*-----------------------------------------------------------------PULSANTIERE----------------------------------------------------------------------------------*)

(**************variabili utilizzate nella logica di controllo (e nella simulazione)***************)

(* PULSANTIERA DI COMANDO*)

	Start:BOOL; (*Pulsante di start*)
	LightStart:BOOL; (*Luce del pulsante di start*)
	Reset:BOOL; (*Pulsante di reset*)
	LightReset:BOOL; (*Luce del pulsante di reset*)
	Stop:BOOL:=TRUE; (*Pulsante di stop*)
	FreezeStop:BOOL:=TRUE; (*Pulsate di "congelamento" del sistema*)
	EmergencyStop:BOOL:=TRUE; (*Pulsante di stop di emergenza*)
	FreezeStopPuls:BOOL:=TRUE; (*Pulsate di "congelamento" del sistema*)

(* PULSANTIERA DI CONTROLLO*)

	LightEmptyWarehouse: BOOL; (*Luce magazzino basi vuoto*)
	FullWarehouse:BOOL; (*Pulsante magazzino basi riempito*)
	LightUpsideDownLoadInExpelling:BOOL; (*Luce pezzo capovolto*)
	LightEmptyCoverHouse:BOOL; (*Luce magazzino coperchi vuoto*)
	FullWarehouseInAssemblyStation:BOOL; (*Pulsante magazzino coperchi riempito*)
	ToWorkBlackLoad:BOOL; (*Selettore colore pezzi da lavorare*)
	ToWorkBlackOrRedLoad:BOOL := TRUE; (*Selettore tipo pezzi da lavorare*)
	UpsideDownLoadRemovedInExpelling:BOOL; (*Pulsante pezzo capovolto rimosso*)
	LightRobotInMovement:BOOL; (*Luce robot in movimento*)
	LightRobotServoON:BOOL; (*Luce motori robot accesi*)
	LightRedLoad:BOOL; (*Luce pezzo rosso/metallico*)
	LightBlackLoad:BOOL; (*Luce pezzo nero*)

(************************************************************************************************)

(* VARIABILI ASSOCIATE ALLE PULSANTIERE ---------solo per la simulazione--------*)

(*pulsantiera virtuale*)
	ToWorkBlackLoadPuls: BOOL;
	ToWorkBlackOrRedLoadPuls: BOOL;
	FullWarehousePuls: BOOL;
	UpsideDownLoadRemovedInExpellingPuls:BOOL;
	FullWarehouseInAssemblyStationPuls: BOOL;
	EnableVirtualBox: BOOL := TRUE; (*pulsante di abilitazione pulsantiera virtuale (disabilitazione pulsantiera fisica)*)
	Remove: BOOL; (*pulsante di rimozione di tutti i pezzi dall'impianto*)

(*pulsantiera fisica*)
	ToWorkBlackLoadPin: BOOL;
	ToWorkBlackOrRedLoadPin: BOOL;
	FullWarehousePin: BOOL;
	UpsideDownLoadRemovedInExpellingPin:BOOL;
	FullWarehouseInAssemblyStationPin: BOOL;

(*-----------------------------------------------------------------------------------------------------------------------------------------------------------*)
(*---------------------------------------------------------------------GUASTI---------------------------------------------------------------------------*)

(* --------------------SIMULAZIONE guasti--------------------- *)

(****variabili utilizzate solo per la simulazione****)

(*MODULO MAGAZZINO DI STOCCAGGIO (magazzion basi)*)

(*sensori: possono essere bloccati alti (a 1) o bloccati bassi (a 0)*)
	EmptyWarehouseBlockHigh: BOOL;
	EmptyWarehouseBlockLow: BOOL;
	CylinderExtractionLoadInRetroactivePositionBlockLow: BOOL;
	CylinderExtractionLoadInRetroactivePositionBlockHigh: BOOL;
	CylinderExtractionLoadInExtensivePositionBlockLow: BOOL;
	CylinderExtractionLoadInExtensivePositionBlockHigh: BOOL;
(*attuatori: possono essere bloccati o bloccato alti (a 1)*)
	CylinderExtractsLoadFromWarehouseBlock: BOOL;
	CylinderExtractsLoadFromWarehouseBlockHigh: BOOL;

(* MODULO DI TRASFERIMENTO (braccio rotante) *)

(*sensori: possono essere bloccati alti (a 1) o bloccati bassi (a 0)*)
	VacuumGeneratorOkBlockHigh: BOOL;
	VacuumGeneratorOkBlockLow: BOOL;
	RotaryMakerInPositionWarehouseBlockHigh: BOOL;
	RotaryMakerInPositionWarehouseBlockLow: BOOL;
	RotaryMakerInPositionVerificationBlockHigh: BOOL;
	RotaryMakerInPositionVerificationBlockLow: BOOL;

(*attuatori: possono essere bloccati o bloccati alti (a 1)*)
	VacuumGeneratorBlock: BOOL;
	VacuumGeneratorBlockHigh: BOOL;
	ExpulsionAirVacuumBlock: BOOL;
	ExpulsionAirVacuumBlockHigh: BOOL;
	RotaryMakerVsWarehouseBlock: BOOL;
	RotaryMakerVsWarehouseBlockHigh: BOOL;
	RotaryMakerVsVerificationBlock: BOOL;
	RotaryMakerVsVerificationBlockHigh: BOOL;

(* STAZIONE DI VERIFICA *)

(*sensori: possono essere bloccati alti (a 1) o bloccati bassi (a 0)*)
	VerificationBusyBlockLow: BOOL;
	VerificationBusyBlockHigh: BOOL;
	ReadyLoadForVerificationBlockHigh: BOOL;
	ReadyLoadForVerificationBlockLow: BOOL;
	CylinderDownToMeasureLoadBlockHigh: BOOL;
	CylinderDownToMeasureLoadBlockLow: BOOL;
	CylinderUpToMeasureLoadBlockHigh: BOOL;
	CylinderUpToMeasureLoadBlockLow: BOOL;
	CylinderOfExtractionInRetroactivePositionBlockHigh: BOOL;
	CylinderOfExtractionInRetroactivePositionBlockLow: BOOL;
	ColourMeasurementBlockHigh: BOOL;
	ColourMeasurementBlockLow: BOOL;
	MeasurementNotOkBlockHigh: BOOL;
	MeasurementNotOkBlockLow: BOOL;

(*attuatori: possono essere bloccati o bloccati alti (a 1)*)
	ToLiftCylinderToMeasureLoadBlock: BOOL;
	ToLiftCylinderToMeasureLoadBlockHigh: BOOL;
	ToLowerCylinderToMeasureLoadBlock: BOOL;
	ToLowerCylinderToMeasureLoadBlockHigh: BOOL;
	ToExtendCylinderOfExtractionVsGuideBlock: BOOL;
	ToExtendCylinderOfExtractionVsGuideBlockHigh: BOOL;
	AirCushionBlock: BOOL;
	AirCushionBlockHigh: BOOL;


(*-------------------------RILEVAZIONE guasti ---------------------------*)

(************variabili utilizzate nella logica di controllo (e nella simulazione)***********)

(* MODULO MAGAZZINO DI STOCCAGGIO (magazzion basi) *)

(*sensori: possono essere bloccati alti (a 1) o bloccati bassi (a 0)*)
	EmptyWarehouseBlockedHigh: BOOL;
	EmptyWarehouseBlockedLow: BOOL;
	CylinderExtractionLoadInRetroactivePositionBlockedLow: BOOL;
	CylinderExtractionLoadInRetroactivePositionBlockedHigh: BOOL;
	CylinderExtractionLoadInExtensivePositionBlockedLow: BOOL;
	CylinderExtractionLoadInExtensivePositionBlockedHigh: BOOL;

(*attuatori: possono essere bloccati o bloccati alti (a 1)*)
	CylinderExtractsLoadFromWarehouseBlocked: BOOL;
	CylinderExtractsLoadFromWarehouseBlockedHigh: BOOL;

(* MODULO DI TRASFERIMENTO (braccio rotante) *)

(*sensori: possono essere bloccati alti (a 1) o bloccati bassi (a 0)*)
	VacuumGeneratorOkBlockedHigh: BOOL;
	VacuumGeneratorOkBlockedLow: BOOL;
	RotaryMakerInPositionWarehouseBlockedHigh: BOOL;
	RotaryMakerInPositionWarehouseBlockedLow: BOOL;
	RotaryMakerInPositionVerificationBlockedHigh: BOOL;
	RotaryMakerInPositionVerificationBlockedLow: BOOL;

(*attuatori: possono essere bloccati o bloccati alti (a 1)*)
	VacuumGeneratorBlocked: BOOL;
	VacuumGeneratorBlockedHigh:BOOL;
	ExpulsionAirVacuumBlocked: BOOL;
	ExpulsionAirVacuumBlockedHigh:BOOL;
	RotaryMakerVsWarehouseBlocked: BOOL;
	RotaryMakerVsWarehouseBlockedHigh: BOOL;
	RotaryMakerVsVerificationBlocked: BOOL;
	RotaryMakerVsVerificationBlockedHigh: BOOL;

(* STAZIONE DI VERIFICA *)

(*sensori: possono essere bloccati alti (a 1) o bloccati bassi (a 0)*)
	VerificationBusyBlockedLow: BOOL;
	VerificationBusyBlockedHigh: BOOL;
	ReadyLoadForVerificationBlockedHigh: BOOL;
	ReadyLoadForVerificationBlockedLow: BOOL;
	CylinderDownToMeasureLoadBlockedHigh: BOOL;
	CylinderDownToMeasureLoadBlockedLow: BOOL;
	CylinderUpToMeasureLoadBlockedHigh: BOOL;
	CylinderUpToMeasureLoadBlockedLow: BOOL;
	CylinderOfExtractionInRetroactivePositionBlockedHigh: BOOL;
	CylinderOfExtractionInRetroactivePositionBlockedLow: BOOL;
	ColourMeasurementBlockedHigh: BOOL;
	ColourMeasurementBlockedLow: BOOL;
	MeasurementNotOkBlockedHigh: BOOL;
	MeasurementNotOkBlockedLow: BOOL;

(*attuatori: possono essere bloccati o bloccati alti (a 1)*)
	ToLiftCylinderToMeasureLoadBlocked: BOOL;
	ToLiftCylinderToMeasureLoadBlockedHigh:BOOL;
	ToLowerCylinderToMeasureLoadBlocked: BOOL;
	ToLowerCylinderToMeasureLoadBlockedHigh: BOOL;
	ToExtendCylinderOfExtractionVsGuideBlocked: BOOL;
	ToExtendCylinderOfExtractionVsGuideBlockedHigh:BOOL;
	AirCushionBlocked: BOOL;
	AirCushionBlockedHigh:BOOL;

(*---------------------------------------------------------------------------------------------------------------------------------*)
(* ALTRE VARIABILI IMPIEGATE NELLA LOGICA DI CONTROLLO (e utilizzate anche nella simulazione) *)

	UncorrectComparison: BOOL; (*comparazione tra l'altezza del pezzo e il colore rilevato: 1 se la misura è incompatibile con il colore, 0 altrimenti*)
	VirtualCylinderDownToMeasureLoad: BOOL; (*sensore virtuale finecorsa inferiore ascensore. Quando l'ascensore scende, va a 1 sul secondo fronte di discesa del sensore CylinderDownToMeasureLoad*)




	(*variabili di controllo utilizzate dalla mia politica di controllo*)
	Stopped: BOOL;
	EndInit: BOOL; (*fine inizializzazione*)
	EndAssembling: BOOL;
	EndProcessing: BOOL;
	EmptyCover: BOOL;

																	(*VARIABILI DI SIMULAZIONE*)
(*___________________________________________________________________________________________________________________________________________*)



	(*VARIABILI DI INIZIALIZZAZIONE CASUALE DELLE GRANDEZZE DEGLI ATTUATORI NON PNEUMATICI*)
	RotaryVisIn: INT;
	DrillingUnitHeight: INT;



	(*STAZIONE DI LAVORAZIONE*)

	(* MODULO TAVOLA ROTANTE*)
	RotaryTablePosition:INT; (*VARIABILE DI VISUALIZZAZIONE:  incremento della posizione della tavola(resettata al primo allineamento) *)
	RotaryTableVisual:INT; (*VARIABILE DI VISUALIZZAZIONE:  incremento della posizione della tavola(con offset iniziale)*)
	Alligneed: BOOL; (*VARIABILE DI SIMULAZIONE:  indica l'allineamento della tavola*)

	(*VARIABILI PER LA GESTIONE DEI COLORI DEI PEZZI NELLE STAZIONI DELLA GIOSTRA*)

	(*                                                                              NERO            BIANCO              ROSSO                GRIGIO     *)
	ColorCircle : ARRAY[1..4] OF DWORD := 16#00000000,16#00FFFFFF, 16#000000FF, 16#00E1E1E1;
	Color1: DWORD:=16#00FFFFFF;
	Color2: DWORD:=16#00FFFFFF;
	Color3: DWORD:=16#00FFFFFF;
	Color4: DWORD:=16#00FFFFFF;
	Color5: DWORD:=16#00FFFFFF;
	Color6: DWORD:=16#00FFFFFF;

	ElementOneTableCharged:BOOL;
	ElementOneTableRed:BOOL;
	ElementOneTableBlack:BOOL;
	ElementOneTableSilver:BOOL;
	ElementOneTableOverturned:BOOL;
	LinearTablePosition1: LREAL;

	ElementTwoTableCharged: BOOL;
	ElementTwoTableRed:BOOL;
	ElementTwoTableBlack:BOOL;
	ElementTwoTableSilver:BOOL;
	ElementTwoTableOverturned:BOOL;
	LinearTablePosition2:LREAL;

	ElementThreeTableCharged:BOOL;
	ElementThreeTableRed:BOOL;
	ElementThreeTableBlack:BOOL;
	ElementThreeTableSilver:BOOL;
	ElementThreeTableOverturned:BOOL;
	LinearTablePosition3: LREAL;

	ElementFourTableCharged: BOOL;
	ElementFourTableRed:BOOL;
	ElementFourTableBlack:BOOL;
	ElementFourTableSilver:BOOL;
	ElementFourTableOverturned:BOOL;
	LinearTablePosition4:LREAL;

	ElementFiveTableCharged:BOOL;
	ElementFiveTableRed:BOOL;
	ElementFiveTableBlack:BOOL;
	ElementFiveTableSilver:BOOL;
	ElementFiveTableOverturned:BOOL;
	LinearTablePosition5: LREAL;

	ElementSixTableCharged: BOOL;
	ElementSixTableRed:BOOL;
	ElementSixTableBlack:BOOL;
	ElementSixTableSilver:BOOL;
	ElementSixTableOverturned:BOOL;
	LinearTablePosition6:LREAL;

	(*VARIABILI PER VISUALIZZARE 'O' SE IL PEZZO E' OVERTURNED*)
	ElementOneTableO: STRING;
	ElementTwoTableO: STRING;
	ElementThreeTableO: STRING;
	ElementFourTableO: STRING;
	ElementFiveTableO: STRING;
	ElementSixTableO: STRING;
	ElementSleighO: STRING;
	ElementStation1RobotO: STRING;

	(* MODULO DI CONTROLLO*)
	InspectPosition:INT; (*VARIABILE DI VISUALIZZAZIONE: incremento posizione utensile per il controllo*)
	InspectDepth: INT; (*variabile utilizzata per simulare le 2 differenti profondità a cui si porta l'utensile di controllo in caso di base corretta o di base Overturned*)
	FLAGInControlLoadInWrongPositionToBeDrilled: BOOL; (*variabile utilizzata per mantenere acceso il led del sensore "InControlLoadInWrongPositionToBeDrilled" in caso di bloccaggio alto*)
      	(* MODULO DI FORATURA.*)
	DrillingUnitPosition:INT; (*VARIABILE DI VISUALIZZAZIONE: incremento della posizione dell'utensile di foratura*)
	BlockingActuator:INT;(*VARIABILE DI VISUALIZZAZIONE: incremento pistone di bloccaggio*)
	DrillingToolColor: BOOL; (*VARIABILE DI VISUALIZZAZIONE : cambio colore alla punta del trapano quando quest'ultimo viene attivato*)

       (* MODULO DI ESPULSIONE.*)
	AvailableLoadInExpulsionPositioning: BOOL:=FALSE; (*variabile fittizia per segnalare l'arrivo della base nella 4stazione della giostra*)
	LeverPosition:INT:=0; (*VARIABILE DI VISUALIZZAZIONE: incremento rotazione leva*)

	(*Slitta tra lavorazione e assemblaggio*)
	ElementSleighCharged: BOOL;
	ElementSleighRed: BOOL;
	ElementSleighSilver: BOOL;
	ElementSleighBlack: BOOL;
	ElementSleighOverturned:BOOL;
	MovementElementSleigh: INT;


	(*STAZIONE DI ASSEMBLAGGIO*)

	(*Stazione1 della stazione di assemblaggio*)
	ElementStation1RobotCharged: BOOL;
	ElementStation1RobotRed: BOOL;
	ElementStation1RobotBlack: BOOL;
	ElementStation1RobotSilver: BOOL;
	ElementStation1RobotOverturned: BOOL;

	(*STAZIONE DI CONTENIMENTO DEI PEZZI SCARICHI*)
	CanDiscard:BOOL:=FALSE;
	(*visualizzazione della base che finisce nel cesto degli scarti*)
	ElementToDiscard: BOOL;
	ElementToDiscardPosition: INT:=0;
	ElementToDiscardRed: BOOL;
	ElementToDiscardSilver: BOOL;
	ElementToDiscardBlack: BOOL;

	(*STAZIONE DI ASSEMBLAGGIO PEZZO*)
	ElementAssemblyCharged: BOOL;
	ElementAssemblyRed: BOOL;
	ElementAssemblySilver: BOOL;
	ElementAssemblyBlack: BOOL;
	CoverAssembly: BOOL;
	PistonBlackAssembly: BOOL;
	PistonSilverAssembly: BOOL;
	SpringAssembly: BOOL;

 	(* MODULO MOLLE.*)
	VisualSpring:BOOL; (* VARIABILE DI VISUALIZZAZIONE: moto traslatorio molla*)
	Spring1:BOOL;  (* VARIABILE DI VISUALIZZAZIONE: *)
      	Spring2:BOOL;  (* VARIABILE DI VISUALIZZAZIONE: *)
	Spring3:BOOL;  (* VARIABILE DI VISUALIZZAZIONE: *)
	Spring4:BOOL;  (* VARIABILE DI VISUALIZZAZIONE: *)
	Spring5:BOOL;  (*VARIABILE DI VISUALIZZAZIONE: *)
	Spring6:BOOL;  (*VARIABILE DI VISUALIZZAZIONE: *)
	Spring7:BOOL;  (* VARIABILE DI VISUALIZZAZIONE: *)
	Spring8:BOOL; (* VARIABILE DI VISUALIZZAZIONE: *)
	ExtractSpringPosition: INT:=40; (*la molla mantiene il cilindro in posizione di riposo NA*)
	EmptySpringWarehouse: BOOL:=TRUE;
	SpringNumber: INT;
	SpringLoad: BOOL:=FALSE;


	(* MODULO MAGAZZINO  PISTONI.*)
	PistonBlack8: BOOL;
	PistonBlack7: BOOL;
	PistonBlack6: BOOL;
	PistonBlack5: BOOL;
	PistonBlack4: BOOL;
	PistonBlack3: BOOL;
	PistonBlack2: BOOL;
	PistonBlack1: BOOL;
	VisualPistonBlack: BOOL; (*VARIABILE DI VISUALIZZAZIONE: traslazione del pistoncino*)
	PistonBlackNumber:INT;

	PistonSilver1: BOOL;
	PistonSilver2: BOOL;
	PistonSilver3: BOOL;
	PistonSilver4: BOOL;
	PistonSilver5: BOOL;
	PistonSilver6: BOOL;
	PistonSilver7: BOOL;
	PistonSilver8: BOOL;
	VisualPistonSilver: BOOL;
	PistonSilverNumber:INT;

	PistonSelectorPosition: INT:=20;(*VARIABILE DI VISUALIZZAZIONE:  movimento orizzontale del cilindro di estrazione pistoni*)
	VisualPistonBlackPosition: INT;(*VARIABILE DI VISUALIZZAZIONE:  movimento orizzontale del pistone nero*)
	VisualPistonSilverPosition: INT;(*VARIABILE DI VISUALIZZAZIONE:  movimento orizzontale del pistone grigio*)
	PistonLoad: BOOL; (*carica contemporaneamente i pistoni neri e grigi*)
	PistonBlackLoad: BOOL; (*carica pistoni black*)
	PistonSilverLoad: BOOL; (*carica pistoni silver*)
	(* magazzino pistoni nero o rosso vuoto. IN REALTA' NON C'E' ALCUN SENSORE DI PRESENZA*)
	EmptyBlackOrRedPistonWarehouseInAssemblyStation:BOOL:=TRUE;
	EmptyPistonBlackWarehouse: BOOL:=TRUE;
	EmptyPistonSilverWarehouse: BOOL:=TRUE;

	(* MODULO STOCCAGGIO COPERCHI.*)
	VisualCover:BOOL;
	Cover1:BOOL; (* variabile utilizzata per rendere visibile un coperchio nel magazzino cover *)
	Cover2:BOOL; (* variabile utilizzata per rendere visibile un coperchio nel magazzino cover *)
	Cover3:BOOL; (* variabile utilizzata per rendere visibile un coperchio nel magazzino cover *)
	Cover4:BOOL; (* variabile utilizzata per rendere visibile un coperchio nel magazzino cover *)
	Cover5:BOOL; (* variabile utilizzata per rendere visibile un coperchio nel magazzino cover *)
	Cover6:BOOL; (* variabile utilizzata per rendere visibile un coperchio nel magazzino cover *)
	Cover7:BOOL; (* variabile utilizzata per rendere visibile un coperchio nel magazzino cover *)
	Cover8:BOOL; (* variabile utilizzata per rendere visibile un coperchio nel magazzino cover *)
	ExtractCoverPosition: INT:=0;
	CoverLoad: BOOL;
	CoverNumber: INT;

	(* STAZIONE DI ASSEMBLAGGIO PEZZO - MODULO BLOCCAGGIO*)
	BlockingCylinderActiveInAssemblyStation:BOOL; (* cilindro di bloccaggio blocca pezzo *)
	CylinderPositionInAssemblyUnit: INT;

	(* ROBOT.*)
	StopProgramRunning: BOOL; (*VARIABILE DI VISUALIZZAZIONE: associata al pulsante omonimo, simula il bloccaggio del programma CosiRop*)
	RobotGoVerticalPosition: INT:=0; (*VARIABILE DI VISUALIZZAZIONE: incremento di posizione lungo l'asse verticale*)
	RobotGoHorizontalPosition: INT:=0; (*VARIABILE DI VISUALIZZAZIONE: incremento di posizione lungo l'asse orizzontale*)
	RobotProgramRunning: BOOL;
	(*5 bit di output dal PLC al robot, le configurazioni di bit relative alle istruzioni sono implementate nel program(OutputBitConfiguration)*)
	Bit0Output: BOOL;
	Bit1Output: BOOL;
	Bit2Output: BOOL;
	Bit3Output: BOOL;
	Bit4Output: BOOL;
	(*4 bit di input dal robot al PLC, le configurazioni di bit relative ai sensori virtuali sono implementate nel program(OutputBitConfiguration)*)
	Bit0Input: BOOL;
	Bit1Input: BOOL;
	Bit2Input: BOOL;
	Bit3Input: BOOL;

	(*VARIABILI DI VISUALIZZAZIONE: per rendere visibili gli elementi nell'end-effector*)
	EndEffectorPosition: INT:=0; (*VARIABILE DI VISUALIZZAZIONE: incremento di posizione "slide" del end effector*)
	ElementInEndEffectorO: STRING; (*aggiunto, O nella base nell'end-effector*)
	ElementInEndEffector: BOOL; (*aggiunto, rende visibile la base nell'end-effector*)
	ElementInEndEffectorBlack: BOOL;
	ElementInEndEffectorRed: BOOL;
	ElementInEndEffectorSilver: BOOL;
	ElementInEndEffectorOverturned: BOOL;
	PistonBlackInEndEffector: BOOL;
	PistonSilverInEndEffector: BOOL;
	SpringInEndEffector: BOOL;
	CoverInEndEffector: BOOL;

	(*VARIABILI UTILIZZATE PER LO SCAMBIO DI PEZZI TRA END-EFFECTOR E MAGAZZINI*)
	SpringExtract: BOOL;
	PistonSilverExtract: BOOL;
	PistonBlackExtract:BOOL;
	CoverExtract: BOOL;

	(*VARIABILE CHE VIENE MESSA A TRUE QUANDO UN ELEMENTO E' COMPLETAMENTE ASSEMBLATO*)
	ElementAssembled: BOOL;

	(*Variabili per visualizzazione cestino scarti-pezzi finiti*)
	CanColour: BOOL; (*variabile utilizzata per cambiare il colore del cestino a seconda che esso venga utilizzato per gli scarti o per i pezzi finiti*)
	CanText: STRING; (*variabile utilizzata per cambiare il testo nel cestino a seconda che esso venga utilizzato per gli scarti o per i pezzi finiti*)
	CoverToDiscard: BOOL; (*variabile utilizzata per visualizzare il coperchio nella base che finisce nel cestino*)
	ElementToDiscardO: STRING; (*variabile utilizzata per visualizzare la "O" nella base che finisce nel cestino*)
	PistonBlackToDiscard: BOOL; (*variabile utilizzata per visualizzare il pistone nero nella base che finisce nel cestino*)
	PistonSilverToDiscard: BOOL; (*variabile utilizzata per visualizzare il pistone grigio nella base che finisce nel cestino*)


	DisplayText: STRING; (*variabile utilizzata per indicare passo-passo le istruzioni da compiere per un corretto funzionamento del sistema*)
	FillAllWarehouses:BOOL:=FALSE; (*variabile collegata al pulsante, che simula lo riempimento di tutti i magazzini della stazione di assemblaggio*)
	(**************************************************************************************************)


	(*VARIABILI DI SIMULAZIONE DIAGNOSTICA*)
	(*........................................................................................................................*)
	(*SENSORI*)
	AlignementRotaryTableWithPositioningsBlockHigh:BOOL;
	AlignementRotaryTableWithPositioningsBlockLow:BOOL;

	AvailableLoadForWorkingStationBlockHigh:BOOL;
	AvailableLoadForWorkingStationBlockLow:BOOL;

	AvailableLoadInControlPositioningBlockHigh:BOOL;
	AvailableLoadInControlPositioningBlockLow:BOOL;

	AvailableLoadInDrillingPositioningBlockHigh:BOOL;
	AvailableLoadInDrillingPositioningBlockLow:BOOL;

	InControlLoadInWrongPositionToBeDrilledBlockHigh: BOOL;
	InControlLoadInWrongPositionToBeDrilledBlockLow: BOOL;

	DrillingUnitUpBlockHigh: BOOL;
	DrillingUnitUpBlockLow: BOOL;

	DrillingUnitDownBlockHigh: BOOL;
	DrillingUnitDownBlockLow: BOOL;

	AvailableLoadForRobotBlockHigh: BOOL;
	AvailableLoadForRobotBlockLow: BOOL;

	RobotInInitialPositionBlockHigh: BOOL;
	RobotInInitialPositionBlockLow: BOOL;

	RobotInAssemblyUnitBlockHigh: BOOL;
	RobotInAssemblyUnitBlockLow: BOOL;

	RobotInPistonWarehouseBlockHigh: BOOL;
	RobotInPistonWarehouseBlockLow: BOOL;

	RobotInSpringWarehouseBlockHigh: BOOL;
	RobotInSpringWarehouseBlockLow: BOOL;

	RobotInCoverWarehouseBlockHigh: BOOL;
	RobotInCoverWarehouseBlockLow: BOOL;

	EmptyCoverHouseInAssemblyStationBlockHigh: BOOL;
	EmptyCoverHouseInAssemblyStationBlockLow: BOOL;

	ToExtractCoverInAssemblyStationInRetroactivePositionBlockHigh: BOOL;
	ToExtractCoverInAssemblyStationInRetroactivePositionBlockLow: BOOL;

	ToExtractCoverInAssemblyStationInExtensivePositionBlockHigh: BOOL;
	ToExtractCoverInAssemblyStationInExtensivePositionBlockLow: BOOL;

	PistonSelectorIsOnTheRightBlockHigh: BOOL;
	PistonSelectorIsOnTheRightBlockLow: BOOL;

	PistonSelectorIsOnTheLeftBlockHigh: BOOL;
	PistonSelectorIsOnTheLeftBlockLow: BOOL;

	ToExtractSpringInAssemblyStationInExtensivePositionBlockHigh: BOOL;
	ToExtractSpringInAssemblyStationInExtensivePositionBlockLow: BOOL;

	ToExtractSpringInAssemblyStationInRetroactivePositionBlockHigh: BOOL;
	ToExtractSpringInAssemblyStationInRetroactivePositionBlockLow: BOOL;

	(*  ATTUATORI  *)

	RotaryTableMotorBlockHigh: BOOL;
	RotaryTableMotorBlockLow: BOOL;

	ToLowerCylinderToInspectLoadBlockHigh: BOOL;
	ToLowerCylinderToInspectLoadBlockLow: BOOL;

	DrillingUnitActiveBlockHigh: BOOL;
	DrillingUnitActiveBlockLow: BOOL;

	ToLowerDrillingUnitBlockHigh: BOOL;
	ToLowerDrillingUnitBlockLow: BOOL;

	ToLiftDrillingUnitBlockHigh: BOOL;
	ToLiftDrillingUnitBlockLow: BOOL;

	BlockingCylinderForwardInDrillingPositioningBlockHigh: BOOL;
	BlockingCylinderForwardInDrillingPositioningBlockLow: BOOL;

	ExpellingLeverActiveBlockHigh: BOOL;
	ExpellingLeverActiveBlockLow: BOOL;

	ToExtractSpringInAssemblyStationBlockHigh: BOOL;
	ToExtractSpringInAssemblyStationBlockLow: BOOL;

	PistonSelectorGoOnTheRightBlockHigh: BOOL;
	PistonSelectorGoOnTheRightBlockLow: BOOL;

	PistonSelectorGoOnTheLeftBlockHigh: BOOL;
	PistonSelectorGoOnTheLeftBlockLow: BOOL;

	ToExtractCoverInAssemblyStationForwardBlockHigh: BOOL;
	ToExtractCoverInAssemblyStationForwardBlockLow: BOOL;

	BlockingCylinderForwardInAssemblyStationBlockHigh: BOOL;
	BlockingCylinderForwardInAssemblyStationBlockLow: BOOL;

	RobotTakeBlackLoadBlockHigh: BOOL;
	RobotTakeBlackLoadBlockLow: BOOL;

	RobotTakeRedSilverLoadBlockHigh: BOOL;
	RobotTakeRedSilverLoadBlockLow: BOOL;

	RobotTakeLoadToDiascardBlockHigh: BOOL;
	RobotTakeLoadToDiascardBlockLow: BOOL;

	RobotGoToInitialPositionBlockHigh: BOOL;
	RobotGoToInitialPositionBlockLow: BOOL;

	RobotGoToSpringHouseBlockHigh: BOOL;
	RobotGoToSpringHouseBlockLow: BOOL;

	RobotGoToPistonHouseBlockHigh: BOOL;
	RobotGoToPistonHouseBlockLow: BOOL;

	RobotGoToCoverHouseBlockHigh: BOOL;
	RobotGoToCoverHouseBlockLow: BOOL;

	RobotTakeCurrentLoadToAssemblyBlockHigh: BOOL;
	RobotTakeCurrentLoadToAssemblyBlockLow: BOOL;

	RobotEngineBlockLow: BOOL;


	(*VARIABILI DI RILEVAZIONE DIAGNOSTICA*)
(*--------------------------------------------------------------------------------------------------*)

	(*SENSORI*)

	AlignementRotaryTableWithPositioningsBlockedHigh:BOOL;
	AlignementRotaryTableWithPositioningsBlockedLow:BOOL;

	AvailableLoadForWorkingStationBlockedHigh:BOOL;
	AvailableLoadForWorkingStationBlockedLow:BOOL;

	AvailableLoadInControlPositioningBlockedHigh:BOOL;
	AvailableLoadInControlPositioningBlockedLow:BOOL;

	AvailableLoadInDrillingPositioningBlockedHigh:BOOL;
	AvailableLoadInDrillingPositioningBlockedLow:BOOL;

	InControlLoadInWrongPositionToBeDrilledBlockedHigh: BOOL;
	InControlLoadInWrongPositionToBeDrilledBlockedLow: BOOL;

	DrillingUnitUpBlockedHigh: BOOL;
	DrillingUnitUpBlockedLow: BOOL;

	DrillingUnitDownBlockedHigh: BOOL;
	DrillingUnitDownBlockedLow: BOOL;

	AvailableLoadForRobotBlockedHigh: BOOL;
	AvailableLoadForRobotBlockedLow: BOOL;

	RobotInInitialPositionBlockedHigh: BOOL;
	RobotInInitialPositionBlockedLow: BOOL;

	RobotInAssemblyUnitBlockedHigh: BOOL;
	RobotInAssemblyUnitBlockedLow: BOOL;

	RobotInPistonWarehouseBlockedHigh: BOOL;
	RobotInPistonWarehouseBlockedLow: BOOL;

	RobotInSpringWarehouseBlockedHigh: BOOL;
	RobotInSpringWarehouseBlockedLow: BOOL;

	RobotInCoverWarehouseBlockedHigh: BOOL;
	RobotInCoverWarehouseBlockedLow: BOOL;

	EmptyCoverHouseInAssemblyStationBlockedHigh: BOOL;
	EmptyCoverHouseInAssemblyStationBlockedLow: BOOL;

	ToExtractCoverInAssemblyStationInRetroactivePositionBlockedHigh: BOOL;
	ToExtractCoverInAssemblyStationInRetroactivePositionBlockedLow: BOOL;

	ToExtractCoverInAssemblyStationInExtensivePositionBlockedHigh: BOOL;
	ToExtractCoverInAssemblyStationInExtensivePositionBlockedLow: BOOL;

	PistonSelectorIsOnTheRightBlockedHigh: BOOL;
	PistonSelectorIsOnTheRightBlockedLow: BOOL;

	PistonSelectorIsOnTheLeftBlockedHigh: BOOL;
	PistonSelectorIsOnTheLeftBlockedLow: BOOL;

	ToExtractSpringInAssemblyStationInExtensivePositionBlockedHigh: BOOL;
	ToExtractSpringInAssemblyStationInExtensivePositionBlockedLow: BOOL;

	ToExtractSpringInAssemblyStationInRetroactivePositionBlockedHigh: BOOL;
	ToExtractSpringInAssemblyStationInRetroactivePositionBlockedLow: BOOL;


	(*  ATTUATORI  *)

	RotaryTableMotorBlockedHigh: BOOL;
	RotaryTableMotorBlockedLow: BOOL;

	ToLowerCylinderToInspectLoadBlockedHigh: BOOL;
	ToLowerCylinderToInspectLoadBlockedLow: BOOL;

	DrillingUnitActiveBlockedHigh: BOOL;
	DrillingUnitActiveBlockedLow: BOOL;

	ToLowerDrillingUnitBlockedHigh: BOOL;
	ToLowerDrillingUnitBlockedLow: BOOL;

	ToLiftDrillingUnitBlockedHigh: BOOL;
	ToLiftDrillingUnitBlockedLow: BOOL;

	BlockingCylinderForwardInDrillingPositioningBlockedHigh: BOOL;
	BlockingCylinderForwardInDrillingPositioningBlockedLow: BOOL;

	ExpellingLeverActiveBlockedHigh: BOOL;
	ExpellingLeverActiveBlockedLow: BOOL;

	ToExtractSpringInAssemblyStationBlockedHigh: BOOL;
	ToExtractSpringInAssemblyStationBlockedLow: BOOL;

	PistonSelectorGoOnTheRightBlockedHigh: BOOL;
	PistonSelectorGoOnTheRightBlockedLow: BOOL;

	PistonSelectorGoOnTheLeftBlockedHigh: BOOL;
	PistonSelectorGoOnTheLeftBlockedLow: BOOL;

	ToExtractCoverInAssemblyStationForwardBlockedHigh: BOOL;
	ToExtractCoverInAssemblyStationForwardBlockedLow: BOOL;

	BlockingCylinderForwardInAssemblyStationBlockedHigh: BOOL;
	BlockingCylinderForwardInAssemblyStationBlockedLow: BOOL;

	RobotTakeBlackLoadBlockedHigh: BOOL;
	RobotTakeBlackLoadBlockedLow: BOOL;

	RobotTakeRedSilverLoadBlockedHigh: BOOL;
	RobotTakeRedSilverLoadBlockedLow: BOOL;

	RobotTakeLoadToDiascardBlockedHigh: BOOL;
	RobotTakeLoadToDiascardBlockedLow: BOOL;

	RobotGoToInitialPositionBlockedHigh: BOOL;
	RobotGoToInitialPositionBlockedLow: BOOL;

	RobotGoToSpringHouseBlockedHigh: BOOL;
	RobotGoToSpringHouseBlockedLow: BOOL;

	RobotGoToPistonHouseBlockedHigh: BOOL;
	RobotGoToPistonHouseBlockedLow: BOOL;

	RobotGoToCoverHouseBlockedHigh: BOOL;
	RobotGoToCoverHouseBlockedLow: BOOL;

	RobotTakeCurrentLoadToAssemblyBlockedHigh: BOOL;
	RobotTakeCurrentLoadToAssemblyBlockedLow: BOOL;

	RobotEngineBlockedLow: BOOL;

	RobotProgramRunningBlockedLow: BOOL;

	EndVerification: BOOL;
	Colour: BOOL;
	View: BOOL;

(*Variabili di comunicazione nel main*)
	InitializationFinished: BOOL;
       ReadyLoadForRotaryTable:BOOL:=FALSE;
       ExpelledLoadFromVerification:BOOL:=FALSE;
	LoadInVerification: BOOL;
	VerificationFree: BOOL; (*Indica la fine delle operazioni della stazione di verifica*)
	VirtualSensorConnectionAlignementRotaryTable: BOOL;
      CommunicationLoadInCorrectPosition:BOOL;
	EndRotaryTable: BOOL:=FALSE;   (*Variabile che indica la fine della rotazione della tavola per il timer*)
	ColorCurrentLoad: STRING;
       BufferColor: ARRAY [1..5] OF STRING:='Empty','Empty','Empty','Empty','Empty';(*Posto1:Inizio giostra. Posto2:Stazione di controllo. Posto3:Stazione di foratura. Posto4:Stazione di espulsione. Posto5:Stazione robot*)
       BufferWrongPosition: ARRAY [1..4] OF STRING;(*Posto1:Stazione di controllo. Posto2:Stazione di foratura. Posto3:Stazione di espulsione. Posto4:Stazione robot*)
	RobotRemovedPiston: BOOL;
	ColorVisualization:ARRAY[1..5] OF DWORD:=16#FFFFFF,16#FFFFFF,16#FFFFFF,16#FFFFFF,16#FFFFFF;
	PositionVisualization:ARRAY[1..4] OF DWORD:=16#FFFFFF,16#FFFFFF,16#FFFFFF,16#FFFFFF;
	LoadTransportOK: BOOL;(*Booleana usata per indicare che non c'è stato un problema nel trasporto del pezzo da magazzino a verifica*)

(*Variabili per la visualizzazione della macchina astati*)
	IndicatorStateIdle: BOOL;
	IndicatorStateCheck: BOOL;
	IndicatorStateInit: BOOL;
	IndicatorStateReady: BOOL;
	IndicatorStateRun: BOOL;
	IndicatorStateStop: BOOL;
	IndicatorStateFreeze: BOOL;
	IndicatorStateAlarm: BOOL;
	IndicatorStateSafe: BOOL;
	IndicatorStateReset: BOOL;
	EndCheck: BOOL;
	EndAlarm: BOOL;
	EndSafe: BOOL;
       EndStop1:BOOL;
       EndStop2:BOOL;
	EndFreeze: BOOL;

(*Luci pulsantiera lampeggianti in emergenza*)

	MachineNOTOkForReset: BOOL:=TRUE;   (*Indica se la macchina è piena e tale da no potere fare il reset*)
      TextMachineEmptyForReset:STRING := 'PRESS TO EMPTY MACHINE' ;
	LightMachineToBeEmpty: BOOL := TRUE;
	ButtonMachineToBeEmptyInvisible:BOOL:=FALSE; (*Serve a rendere invisibile il pulsante di richiesta di svuotamento macchina*)
	TypeOfFault: STRING; (*Utilizzata nella visualizzazione per vedere il tipo di guasto rilevato*)
	FaultRemoved: BOOL; (*Pulsante utente per rimuovore l'allarme dovuto a guasti*)
	PossibleFault: BOOL;  (*Utilizzata dal Diagnoser per indicare se è stato rilevata una situazione di possibile guasto. La machina viene fermata in fase*)

(***************************************)
(*****TIMERS DI DIAGNOSTICA******)
(***************************************)

	ExtractionCyliderInActuation: TON; (*Timer cilindro distribuzione in estrazione*)
	ExtractionCyliderInDeactivation: TON; (*Timer cilindro distribuzione in retrazione*)
	ElevatorInUpMovement: TON;  (*Timer elevatore in salita*)
	ElevatorInDownMovement: TON;  (*Timer elevatore in discesa*)
	DiagRotaryTableActivation: TON;   (*Timer tavola rotante in attivazione*)
	DiagRotaryTableDeactivation: TON; (*Timer tavola rotante in disattivazione*)

(*Variabili per l'attivazione dei timer di diagnostica*)

	TimeDiagExtractCylinderInActuation: BOOL; (*Attivazione timer diagnostica estrazione cilindro*)
	TimeDiagExtractCylinderInDeactivation: BOOL; (*Attivazione timer diagnostica retrazione cilindro*)
	TimeDiagElevatorInUpMovement: BOOL; (*Attivazione timer diagnostica elevatore in salita*)
	TimeDiagElevatorInDownMovement: BOOL; (*Attivazione timer diagnostica elevatore in discesa*)
	TimeDiagRotaryTableDeactivation: BOOL;  (*Attivazione timer diagnostica tavola in disattivazione*)
	TimeDiagRotaryTableActivation: BOOL; (*Attivazione timer diagnostica tavola in attivazione*)

(**********************************************************************)
(*****STRINGE DI COMUNICAZIONE MALFUNZIONAMENTI******)
(**********************************************************************)

	ComunicationFaultElevator: STRING; (*Tipo di fault per l'elevatore*)
	ComunicationFaultRotaryTable:STRING; (*Tipo di fault per la tavola rotante*)
	ComunicationFaultExtractionCylinder:STRING; (*Tipo di fault per il cilindro di estrazione*)
       ComunicationFaultSensorPresenceVerification:STRING; (*Tipo di fault per il sensore di presenza in verifica*)

(**********************************************************************)
(*****VARIABILI DELL' INTERFACCIA GRAFICA DI ALLARME******)
(**********************************************************************)
	SensorCylinderExtractFault:BOOL; (*Guasto al finecorsa esteso*)
	SensorCylinderRetractFault:BOOL; (*Guasto al finecorsa retratto*)
	CylinderMovementFault:BOOL; (*Guasto all'attuatore cilindro*)
	SensorElevatorUpFault:BOOL; (*Guasto al finecorsa alto*)
	SensorElevatorDownFault:BOOL; (*Guasto al finecorsa basso*)
	ElevatorMovementFault:BOOL; (*Guasto all'attuatore elevatore*)
	SensorAlignementRotaryTableFault:BOOL; (*Guasto al sensore allineamento tavola*)
	RotaryTableMovementFault:BOOL; (*Guasto all'attuatore tavola*)
	SensorLoadInVerificationFault:BOOL; (*Guasto al sensore presenza in verifica*)
	LoadDroppedByTheCarrierFault:BOOL; (*Guasto pezzo caduto dal braccio rotante*)
	SensorElevatorDownPossibleFault:BOOL; (*Possibile guasto al finecorsa basso*)
END_VAR

(* Global variable list: MyGlobal/TakenFromSimulation *)
VAR_GLOBAL
(*
(******* THOSE VARIABLES ARE ALREADY PRESENT IN "SIM_Global_Var", IF you don't have them UNCOMMENT ****)
	TypeOfFault: STRING; (*Utilizzata nella visualizzazione per vedere il tipo di guasto rilevato*)
	IndicatorStateIdle: BOOL;
	IndicatorStateCheck: BOOL;
	IndicatorStateInit: BOOL;
	IndicatorStateReady: BOOL;
	IndicatorStateRun: BOOL;
	IndicatorStateStop: BOOL;
	IndicatorStateFreeze: BOOL;
	IndicatorStateAlarm: BOOL;
	IndicatorStateSafe: BOOL;
	IndicatorStateReset: BOOL;

	FaultRemoved: BOOL; (*Pulsante utente per rimuovore l'allarme dovuto a guasti*)
	PossibleFault: BOOL;  (*Utilizzata dal Diagnoser per indicare se è stato rilevata una situazione di possibile guasto. La machina viene fermata in fase*)

	MachineNOTOkForReset: BOOL:=TRUE;   (*Indica se la macchina è piena e tale da no potere fare il reset*)
      TextMachineEmptyForReset:STRING := 'PRESS TO EMPTY MACHINE' ;
	LightMachineToBeEmpty: BOOL := TRUE;
	ButtonMachineToBeEmptyInvisible:BOOL:=FALSE; (*Serve a rendere invisibile il pulsante di richiesta di svuotamento macchina*)
*)

	TypeOfFault1: STRING;
	TypeOfFault2: STRING;
	TypeOfFault3: STRING;
	SignalPriorityCode1 : WORD;
	SignalPriorityCode2 : WORD;
	SignalPriorityCode3 : WORD;

	WaitingTime: INT := 10;
	ElementCompleted4: INT;
	ElementRejected4: INT;

END_VAR

(* Data type in MyStructures *)
TYPE CharacterisazionElement :
	STRUCT
		Color:BOOL;
		Over:BOOL := FALSE;
	END_STRUCT
END_TYPE

(* Data type in MyStructures *)
TYPE
	DeviceStateType : 
		(
		DeviceDisabledState := 0,
		DeviceEnablePhaseState,
		DeviceEnabledState,
		DeviceDisablePhaseState
		);
END_TYPE

(* POU 0_Simulation/Pulsantiera, ST *)
PROGRAM Pulsantiera
VAR
END_VAR
(* Pulsantiera di controllo *)
(*IF EnableVirtualBox THEN  (* se la pulsantiera virtuale è abilitata le uscite saranno quelle della pulsantiera virtuale *)
	ToWorkBlackLoad:=ToWorkBlackLoadPuls;
	ToWorkBlackOrRedLoad:=ToWorkBlackOrRedLoadPuls;
	FullWarehouse:=FullWarehousePuls;
	UpsideDownLoadRemovedInExpelling:=UpsideDownLoadRemovedInExpellingPuls;
	FullWarehouseInAssemblyStation:=FullWarehouseInAssemblyStationPuls;
ELSE (*altrimenti uso la pulsantiera fisica*)
	ToWorkBlackLoad:=ToWorkBlackLoadPin;
	ToWorkBlackOrRedLoad:=ToWorkBlackOrRedLoadPin;
	FullWarehouse:=FullWarehousePin;
	UpsideDownLoadRemovedInExpelling:=UpsideDownLoadRemovedInExpellingPin;
	FullWarehouseInAssemblyStation:=FullWarehouseInAssemblyStationPin;
END_IF;
*)
IF FaultDetected
THEN
	(*SENSORI*)
	AlignementRotaryTableWithPositioningsBlockHigh:=FALSE;
	AlignementRotaryTableWithPositioningsBlockLow:=FALSE;

	AvailableLoadForWorkingStationBlockHigh:=FALSE;
	AvailableLoadForWorkingStationBlockLow:=FALSE;

	AvailableLoadInControlPositioningBlockHigh:=FALSE;
	AvailableLoadInControlPositioningBlockLow:=FALSE;

	AvailableLoadInDrillingPositioningBlockHigh:=FALSE;
	AvailableLoadInDrillingPositioningBlockLow:=FALSE;

	InControlLoadInWrongPositionToBeDrilledBlockHigh:=FALSE;
	InControlLoadInWrongPositionToBeDrilledBlockLow:=FALSE;

	DrillingUnitUpBlockHigh:=FALSE;
	DrillingUnitUpBlockLow:=FALSE;

	DrillingUnitDownBlockHigh:=FALSE;
	DrillingUnitDownBlockLow:=FALSE;

	AvailableLoadForRobotBlockHigh:=FALSE;
	AvailableLoadForRobotBlockLow:=FALSE;

	RobotInInitialPositionBlockHigh:=FALSE;
	RobotInInitialPositionBlockLow:=FALSE;

	RobotInAssemblyUnitBlockHigh:=FALSE;
	RobotInAssemblyUnitBlockLow:=FALSE;

	RobotInPistonWarehouseBlockHigh:=FALSE;
	RobotInPistonWarehouseBlockLow:=FALSE;

	RobotInSpringWarehouseBlockHigh:=FALSE;
	RobotInSpringWarehouseBlockLow:=FALSE;

	RobotInCoverWarehouseBlockHigh:=FALSE;
	RobotInCoverWarehouseBlockLow:=FALSE;

	EmptyCoverHouseInAssemblyStationBlockHigh:=FALSE;
	EmptyCoverHouseInAssemblyStationBlockLow:=FALSE;

	ToExtractCoverInAssemblyStationInRetroactivePositionBlockHigh:=FALSE;
	ToExtractCoverInAssemblyStationInRetroactivePositionBlockLow:=FALSE;

	ToExtractCoverInAssemblyStationInExtensivePositionBlockHigh:=FALSE;
	ToExtractCoverInAssemblyStationInExtensivePositionBlockLow:=FALSE;

	PistonSelectorIsOnTheRightBlockHigh:=FALSE;
	PistonSelectorIsOnTheRightBlockLow:=FALSE;

	PistonSelectorIsOnTheLeftBlockHigh:=FALSE;
	PistonSelectorIsOnTheLeftBlockLow:=FALSE;

	ToExtractSpringInAssemblyStationInExtensivePositionBlockHigh:=FALSE;
	ToExtractSpringInAssemblyStationInExtensivePositionBlockLow:=FALSE;

	ToExtractSpringInAssemblyStationInRetroactivePositionBlockHigh:=FALSE;
	ToExtractSpringInAssemblyStationInRetroactivePositionBlockLow:=FALSE;

	(*  ATTUATORI  *)

	RotaryTableMotorBlockHigh:=FALSE;
	RotaryTableMotorBlockLow:=FALSE;

	ToLowerCylinderToInspectLoadBlockHigh:=FALSE;
	ToLowerCylinderToInspectLoadBlockLow:=FALSE;

	DrillingUnitActiveBlockHigh:=FALSE;
	DrillingUnitActiveBlockLow:=FALSE;

	ToLowerDrillingUnitBlockHigh:=FALSE;
	ToLowerDrillingUnitBlockLow:=FALSE;

	ToLiftDrillingUnitBlockHigh:=FALSE;
	ToLiftDrillingUnitBlockLow:=FALSE;

	BlockingCylinderForwardInDrillingPositioningBlockHigh:=FALSE;
	BlockingCylinderForwardInDrillingPositioningBlockLow:=FALSE;

	ExpellingLeverActiveBlockHigh:=FALSE;
	ExpellingLeverActiveBlockLow:=FALSE;

	ToExtractSpringInAssemblyStationBlockHigh:=FALSE;
	ToExtractSpringInAssemblyStationBlockLow:=FALSE;

	PistonSelectorGoOnTheRightBlockHigh:=FALSE;
	PistonSelectorGoOnTheRightBlockLow:=FALSE;

	PistonSelectorGoOnTheLeftBlockHigh:=FALSE;
	PistonSelectorGoOnTheLeftBlockLow:=FALSE;

	ToExtractCoverInAssemblyStationForwardBlockHigh:=FALSE;
	ToExtractCoverInAssemblyStationForwardBlockLow:=FALSE;

	BlockingCylinderForwardInAssemblyStationBlockHigh:=FALSE;
	BlockingCylinderForwardInAssemblyStationBlockLow:=FALSE;

	RobotTakeBlackLoadBlockHigh:=FALSE;
	RobotTakeBlackLoadBlockLow:=FALSE;

	RobotTakeRedSilverLoadBlockHigh:=FALSE;
	RobotTakeRedSilverLoadBlockLow:=FALSE;

	RobotTakeLoadToDiascardBlockHigh:=FALSE;
	RobotTakeLoadToDiascardBlockLow:=FALSE;

	RobotGoToInitialPositionBlockHigh:=FALSE;
	RobotGoToInitialPositionBlockLow:=FALSE;

	RobotGoToSpringHouseBlockHigh:=FALSE;
	RobotGoToSpringHouseBlockLow:=FALSE;

	RobotGoToPistonHouseBlockHigh:=FALSE;
	RobotGoToPistonHouseBlockLow:=FALSE;

	RobotGoToCoverHouseBlockHigh:=FALSE;
	RobotGoToCoverHouseBlockLow:=FALSE;

	RobotTakeCurrentLoadToAssemblyBlockHigh:=FALSE;
	RobotTakeCurrentLoadToAssemblyBlockLow:=FALSE;

	RobotEngineBlockLow:=FALSE;
END_IF;
END_PROGRAM

(* POU 0_Simulation/PlantCarico, ST *)
PROGRAM PlantCarico
VAR
	EstrazioneRosso: INT:=0; (*variabile che memorizza la posizione dei pezzi rossi estratti*)
	EstrazioneSilver:INT:=0; (*variabile che memorizza la posizione dei pezzi argentati estratti*)
	EstrazioneNero: INT:=0; (*variabile che memorizza la posizione dei pezzi neri estratti*)
END_VAR
(*Per caricare gli oggetti nel magazzino, utilizzo un'istruzione "case of" per ogni pulsante -red, silver, black-*)

IF (NOT ElementOneCharged AND (Red OR Redoverturned )) THEN
	EstrazioneRosso:=1 ;(*carico il primo elemento rosso*)
END_IF;

IF (ElementOneCharged AND (Red OR Redoverturned)) THEN
	EstrazioneRosso:=2;
END_IF; (*carico il secondo elemento rosso*)

IF ( ElementTwoCharged  AND (Red OR Redoverturned) ) THEN
	EstrazioneRosso:=3;(*carico il terzo  elemento rosso*)
END_IF;

 IF (ElementThreeCharged AND (Red OR Redoverturned) ) THEN
	EstrazioneRosso:=4;  (*carico il quarto elemento rosso*)
END_IF;

IF (ElementFourCharged AND (Red OR Redoverturned) ) THEN
	EstrazioneRosso:=5; (*carico il quinto elemento rosso*)
END_IF;

IF (ElementFiveCharged AND (Red OR Redoverturned) ) THEN
	EstrazioneRosso:=6;  (*carico il sesto elemento rosso*)
END_IF;

IF (ElementSixCharged AND (Red  OR Redoverturned)) THEN
	EstrazioneRosso:=7; (*carico il settimo elemento rosso*)
END_IF;

IF (ElementSevenCharged AND (Red OR Redoverturned)) THEN
	EstrazioneRosso:=8;  (*carico l'ottavo elemento rosso*)
END_IF;

CASE EstrazioneRosso OF	(*Ogni stato dell'istruzione "case of" corrisponde ad una base*)

1:	ElementOneRed:=TRUE;
	EmptyWarehouse:=FALSE;
	ElementOneCharged:=TRUE;
	Red:=FALSE;
	IF Redoverturned THEN
		ElementOneOverturned:=TRUE;
	END_IF;
	Redoverturned:=FALSE;
	EstrazioneRosso:=0;

2:	ElementTwoRed:=TRUE;
	ElementTwoCharged:=TRUE;
	Red:=FALSE;
	IF   Redoverturned THEN
		ElementTwoOverturned:=TRUE;
	END_IF;
	Redoverturned:=FALSE;
	EstrazioneRosso:=0;

3:	ElementThreeRed:=TRUE;
	ElementThreeCharged:=TRUE;
	Red:=FALSE;
	IF Redoverturned THEN
		ElementThreeOverturned:=TRUE;
	END_IF;
	Redoverturned:=FALSE;
	EstrazioneRosso:=0;

4:	ElementFourRed:=TRUE;
	ElementFourCharged:=TRUE;
	Red:=FALSE;
	IF Redoverturned THEN
		ElementFourOverturned:=TRUE;
	END_IF;
	Redoverturned:=FALSE;
	EstrazioneRosso:=0;

5:	ElementFiveRed:=TRUE;
	ElementFiveCharged:=TRUE;
	Red:=FALSE;
	IF Redoverturned THEN
		ElementFiveOverturned:=TRUE;
	END_IF;
	Redoverturned:=FALSE;
	EstrazioneRosso:=0;

6:	ElementSixRed:=TRUE;
	ElementSixCharged:=TRUE;
	Red:=FALSE;
	IF Redoverturned THEN
		ElementSixOverturned:=TRUE;
	END_IF;
	Redoverturned:=FALSE;
	EstrazioneRosso:=0;

7:	ElementSevenRed:=TRUE;
	ElementSevenCharged:=TRUE;
	Red:=FALSE;
      IF Redoverturned THEN
		ElementSevenOverturned:=TRUE;
	END_IF;
	Redoverturned:=FALSE;
	EstrazioneRosso:=0;

8:	ElementEightRed:=TRUE;
	ElementEightCharged:=TRUE;
	Red:=FALSE;
	IF Redoverturned THEN
		ElementEightOverturned:=TRUE;
	END_IF;
	Redoverturned:=FALSE;
	EstrazioneRosso:=0;
END_CASE;


IF (NOT ElementOneCharged AND (Silver OR Silveroverturned OR Silvershort)) THEN
	EstrazioneSilver:=1 ;
END_IF;

IF (ElementOneCharged  AND (Silver OR Silveroverturned OR Silvershort ) ) THEN
	EstrazioneSilver:=2;
END_IF;

IF ( ElementTwoCharged  AND (Silver OR Silveroverturned  OR Silvershort) ) THEN
	EstrazioneSilver:=3;
END_IF;

 IF (ElementThreeCharged AND (Silver OR Silveroverturned  OR Silvershort) ) THEN
	EstrazioneSilver:=4;
END_IF;

IF (ElementFourCharged AND (Silver OR Silveroverturned  OR Silvershort) ) THEN
	EstrazioneSilver:=5;
END_IF;

IF (ElementFiveCharged AND (Silver OR Silveroverturned  OR Silvershort) ) THEN
	EstrazioneSilver:=6;
END_IF;

IF (ElementSixCharged AND (Silver OR Silveroverturned  OR Silvershort)  ) THEN
	EstrazioneSilver:=7;
END_IF;

IF (ElementSevenCharged AND (Silver OR Silveroverturned  OR Silvershort) ) THEN
		EstrazioneSilver:=8;
END_IF;


CASE EstrazioneSilver OF

1:	ElementOneSilver:=TRUE;
	ElementOneCharged:=TRUE;
	Silver:=FALSE;
	IF Silveroverturned THEN  (* cilindro capovolto *)
		ElementOneOverturned:=TRUE;
	END_IF;
	Silveroverturned:=FALSE;
	IF Silvershort THEN  (* cilindro corto *)
		ElementOneShort:=TRUE;
	END_IF;
	Silvershort:=FALSE;
	EstrazioneSilver:=0;

2:	ElementTwoSilver:=TRUE;
	ElementTwoCharged:=TRUE;
	Silver:=FALSE;
	IF 	Silveroverturned THEN
		ElementTwoOverturned:=TRUE;
	END_IF;
	Silveroverturned:=FALSE;
	IF Silvershort THEN
		ElementTwoShort:=TRUE;
	END_IF;
	Silvershort:=FALSE;
	EstrazioneSilver:=0;

3:	ElementThreeSilver:=TRUE;
	ElementThreeCharged:=TRUE;
	Silver:=FALSE;
	IF Silveroverturned THEN
		ElementThreeOverturned:=TRUE;
	END_IF;
	Silveroverturned:=FALSE;
	IF Silvershort THEN
		ElementThreeShort:=TRUE;
	END_IF;
	Silvershort:=FALSE;
	EstrazioneSilver:=0;

4:	ElementFourSilver:=TRUE;
	ElementFourCharged:=TRUE;
	Silver:=FALSE;
	IF Silveroverturned THEN
		ElementFourOverturned:=TRUE;
	END_IF;
	Silveroverturned:=FALSE;
	IF Silvershort THEN
		ElementFourShort:=TRUE;
	END_IF;
	Silvershort:=FALSE;
	EstrazioneSilver:=0;

5:	ElementFiveSilver:=TRUE;
	ElementFiveCharged:=TRUE;
	Silver:=FALSE;
	IF Silveroverturned THEN
		ElementFiveOverturned:=TRUE;
	END_IF;
	Silveroverturned:=FALSE;
	IF Silvershort THEN
		ElementFiveShort:=TRUE;
	END_IF;
	Silvershort:=FALSE;
	EstrazioneSilver:=0;

6:	ElementSixSilver:=TRUE;
	ElementSixCharged:=TRUE;
	Silver:=FALSE;
	IF Silveroverturned THEN
		ElementSixOverturned:=TRUE;
	END_IF;
	Silveroverturned:=FALSE;
	IF Silvershort THEN
		ElementSixShort:=TRUE;
	END_IF;
	Silvershort:=FALSE;
	EstrazioneSilver:=0;

7:	ElementSevenSilver:=TRUE;
	ElementSevenCharged:=TRUE;
	Silver:=FALSE;
	IF Silveroverturned THEN
		ElementSevenOverturned:=TRUE;
	END_IF;
	Silveroverturned:=FALSE;
	IF Silvershort THEN
		ElementSevenShort:=TRUE;
	END_IF;
	Silvershort:=FALSE;
	EstrazioneSilver:=0;

8:	ElementEightSilver:=TRUE;
	ElementEightCharged:=TRUE;
	Silver:=FALSE;
	IF Silveroverturned THEN
		ElementEightOverturned:=TRUE;
	END_IF;
	Silveroverturned:=FALSE;
	IF Silvershort THEN
		ElementEightShort:=TRUE;
	END_IF;
	Silvershort:=FALSE;
	EstrazioneSilver:=0;
END_CASE;

IF (NOT ElementOneCharged AND (Black OR Blackoverturned) ) THEN
	EstrazioneNero:=1 ;
END_IF;

IF (ElementOneCharged  AND (Black OR Blackoverturned) ) THEN
	EstrazioneNero:=2;
END_IF;

IF ( ElementTwoCharged  AND (Black OR Blackoverturned) ) THEN
	EstrazioneNero:=3;
END_IF;

 IF (ElementThreeCharged AND (Black OR Blackoverturned) ) THEN
	EstrazioneNero:=4;
END_IF;

IF (ElementFourCharged AND (Black OR Blackoverturned)  ) THEN
	EstrazioneNero:=5;
END_IF;

IF (ElementFiveCharged AND (Black OR Blackoverturned) ) THEN
	EstrazioneNero:=6;
END_IF;
IF (ElementSixCharged AND (Black OR Blackoverturned)  ) THEN
	EstrazioneNero:=7;
END_IF;

IF (ElementSevenCharged AND (Black OR Blackoverturned) ) THEN
	EstrazioneNero:=8;
END_IF;


CASE EstrazioneNero OF

1:	ElementOneBlack:=TRUE;
	ElementOneCharged:=TRUE;
	Black:=FALSE;
	IF Blackoverturned THEN
		ElementOneOverturned:=TRUE;
	END_IF;
	Blackoverturned:=FALSE;
	EstrazioneNero:=0;

2:	ElementTwoBlack:=TRUE;
	ElementTwoCharged:=TRUE;
	Black:=FALSE;
	IF Blackoverturned THEN
		ElementTwoOverturned:=TRUE;
	END_IF;
	Blackoverturned:=FALSE;
	EstrazioneNero:=0;

3:	ElementThreeBlack:=TRUE;
	ElementThreeCharged:=TRUE;
	Black:=FALSE;
	IF Blackoverturned THEN
		ElementThreeOverturned:=TRUE;
	END_IF;
	Blackoverturned:=FALSE;
	EstrazioneNero:=0;

4:	ElementFourBlack:=TRUE;
	ElementFourCharged:=TRUE;
	Black:=FALSE;
	IF Blackoverturned THEN
		ElementFourOverturned:=TRUE;
	END_IF;
	Blackoverturned:=FALSE;
	EstrazioneNero:=0;

5:	ElementFiveBlack:=TRUE;
	ElementFiveCharged:=TRUE;
	Black:=FALSE;
	IF Blackoverturned THEN
		ElementFiveOverturned:=TRUE;
	END_IF;
	Blackoverturned:=FALSE;
	EstrazioneNero:=0;

6:	ElementSixBlack:=TRUE;
	ElementSixCharged:=TRUE;
	Black:=FALSE;
	IF Blackoverturned THEN
		ElementSixOverturned:=TRUE;
	END_IF;
	Blackoverturned:=FALSE;
	EstrazioneNero:=0;

7:	ElementSevenBlack:=TRUE;
	ElementSevenCharged:=TRUE;
	Black:=FALSE;
	IF Blackoverturned THEN
		ElementSevenOverturned:=TRUE;
	END_IF;
	Blackoverturned:=FALSE;
	EstrazioneNero:=0;

8:	ElementEightBlack:=TRUE;
	ElementEightCharged:=TRUE;
	Black:=FALSE;
	IF	Blackoverturned THEN
		ElementEightOverturned:=TRUE;
	END_IF;
	Blackoverturned:=FALSE;
	EstrazioneNero:=0;

END_CASE;
END_PROGRAM

(* POU 0_Simulation/PlantScarico, ST *)
PROGRAM PlantScarico
VAR
END_VAR
IF (CylinderBehind AND CylinderPosition<=4) THEN	(*Quando il cilindro di espulsione sta tornando in posizione di riposo, tutti i pezzi ricevono gli attributi dal pezzo che gli e' sopra*)
	ElementOneCharged:=ElementTwoCharged;
	ElementOneRed:=ElementTwoRed;
	ElementOneSilver:=ElementTwoSilver;
	ElementOneBlack:=ElementTwoBlack;
	ElementOneOverturned:=ElementTwoOverturned;
	ElementOneShort:=ElementTwoShort;

	ElementTwoCharged:=ElementThreeCharged;
	ElementTwoRed:=ElementThreeRed;
	ElementTwoSilver:=ElementThreeSilver;
	ElementTwoBlack:=ElementThreeBlack;
	ElementTwoOverturned:=ElementThreeOverturned;
	ElementTwoShort:=ElementThreeShort;

	ElementThreeCharged:=ElementFourCharged;
	ElementThreeRed:=ElementFourRed;
	ElementThreeSilver:=ElementFourSilver;
	ElementThreeBlack:=ElementFourBlack;
	ElementThreeOverturned:=ElementFourOverturned;
	ElementThreeShort:=ElementFourShort;

	ElementFourCharged:=ElementFiveCharged;
	ElementFourRed:=ElementFiveRed;
	ElementFourSilver:=ElementFiveSilver;
	ElementFourBlack:=ElementFiveBlack;
	ElementFourOverturned:=ElementFiveOverturned;
	ElementFourShort:=ElementFiveShort;

	ElementFiveCharged:=ElementSixCharged;
	ElementFiveRed:=ElementSixRed;
	ElementFiveSilver:=ElementSixSilver;
	ElementFiveBlack:=ElementSixBlack;
	ElementFiveOverturned:=ElementSixOverturned;
	ElementFiveShort:=ElementSixShort;

	ElementSixCharged:=ElementSevenCharged;
	ElementSixRed:=ElementSevenRed;
	ElementSixSilver:=ElementSevenSilver;
	ElementSixBlack:=ElementSevenBlack;
	ElementSixOverturned:=ElementSevenOverturned;
	ElementSixShort:=ElementSevenShort;

	ElementSevenCharged:=ElementEightCharged;
	ElementSevenRed:=ElementEightRed;
	ElementSevenSilver:=ElementEightSilver;
	ElementSevenBlack:=ElementEightBlack;
	ElementSevenOverturned:=ElementEightOverturned;
	ElementSevenShort:=ElementEightShort;

 	ElementEightCharged:=FALSE;
	ElementEightRed:=FALSE;
	ElementEightSilver:=FALSE;
	ElementEightBlack:=FALSE;
	ElementEightOverturned:=FALSE;
	ElementEightShort:=FALSE;

END_IF;
END_PROGRAM

(* POU 0_Simulation/PlantMagazzino, ST *)
PROGRAM PlantMagazzino
VAR
	BlockedVsVerification: BOOL; (*flag che segnala il bloccaggio del braccio rotante in posizione verifica*)
	BlockedVsWarehouse: BOOL; (*flag che segnala il bloccaggio del braccio rotante in posizione magazzino*)
END_VAR
(*sensore di presenza pezzo magazzino: *)
IF NOT (EmptyWarehouseBlockHigh OR EmptyWarehouseBlockLow) THEN (*sensore non guasto*)
	IF NOT ElementOneCharged AND NOT ElementTwoCharged THEN (*se non ho elementi caricati in magazzino attivo il sensore*)
			EmptyWarehouse:=TRUE;
		ELSE EmptyWarehouse:=FALSE;
	END_IF;
END_IF;

(*sensore di presenza pezzo magazzino guasto: *)
IF EmptyWarehouseBlockHigh THEN (*bloccato alto*)
	EmptyWarehouse:=TRUE;
END_IF;
IF EmptyWarehouseBlockLow THEN (*bloccato basso*)
	EmptyWarehouse:=FALSE;
END_IF;

(*se il comando di uscita del cilindro e' attivo, e il cilindro non è bloccato, incremento la posizione dello stesso*)
IF NOT (CylinderExtractsLoadFromWarehouseBlock) THEN
	IF CylinderExtractsLoadFromWarehouse AND CylinderPosition<=80 THEN
			CylinderPosition:=CylinderPosition+4;
			ElementPosition:=ElementPosition+4;
		ELSE IF NOT CylinderExtractsLoadFromWarehouse AND CylinderPosition>=0 AND NOT CylinderExtractsLoadFromWarehouseBlockHigh  THEN
				CylinderPosition:=CylinderPosition-4; (*altrimenti, se l'attuatore non è bloccato alto, torna in posizione retratta grazie all'inversione del flusso d'aria*)
				ElementPosition:=0;
			END_IF;
	END_IF;
END_IF;

IF Reset THEN
	CylinderPosition:=0;
END_IF;

(*sensore di finecorsa inferiore cilindro di estrazione: *)
IF (CylinderPosition<1) THEN  (*Controllo che permette al cilindro di mantenersi in posizione di riposo quando non e' attivo il comando di attuazione*)
	CylinderPosition:=0;
	IF NOT (CylinderExtractionLoadInRetroactivePositionBlockHigh OR CylinderExtractionLoadInRetroactivePositionBlockLow) THEN
		CylinderExtractionLoadInRetroactivePosition:=TRUE; (*Sensore attivo quando il cilindro e' in posizione retratta e sensore non gausto*)
	END_IF;
	CylinderBehind:=FALSE; (*Flag vero solo quando il cilindro sta tornardo in posizione di riposo*)
	ELSE IF NOT (CylinderExtractionLoadInRetroactivePositionBlockHigh OR CylinderExtractionLoadInRetroactivePositionBlockLow) THEN
			CylinderExtractionLoadInRetroactivePosition:=FALSE;
		END_IF;
END_IF;

(*sensore di finecorsa inferiore cilindro di estrazione guasto: *)
IF CylinderExtractionLoadInRetroactivePositionBlockHigh THEN
	CylinderExtractionLoadInRetroactivePosition:=TRUE;
END_IF;
IF CylinderExtractionLoadInRetroactivePositionBlockLow THEN
	CylinderExtractionLoadInRetroactivePosition:=FALSE;
END_IF;

IF ElementPosition>=80  THEN
		ElementPosition:=80;
		ReadyForRotaryMaker:=TRUE; (*Quando si trova in posizione "80", il pezzo e' pronto per essere caricato dal RotaryMaker*)
	ELSE
		ReadyForRotaryMaker:=FALSE;
END_IF;

(*sensore di finecorsa superiore cilindro di estrazione: *)
IF CylinderPosition>=80  THEN
	CylinderPosition:=80;
	IF NOT (CylinderExtractionLoadInExtensivePositionBlockHigh OR CylinderExtractionLoadInExtensivePositionBlockLow) THEN
		CylinderExtractionLoadInExtensivePosition:=TRUE; (*Sensore attivo quando il cilindro e' in posizione totalmente estratta e sensore non guasto *)
	END_IF;
	ELSE IF NOT (CylinderExtractionLoadInExtensivePositionBlockHigh OR CylinderExtractionLoadInExtensivePositionBlockLow) THEN
			CylinderExtractionLoadInExtensivePosition:=FALSE;
		END_IF;
END_IF;

(*sensore di finecorsa superiore guasto: *)
IF CylinderExtractionLoadInExtensivePositionBlockHigh THEN
	CylinderExtractionLoadInExtensivePosition:=TRUE;
END_IF;
IF CylinderExtractionLoadInExtensivePositionBlockLow THEN
	CylinderExtractionLoadInExtensivePosition:=FALSE;
END_IF;

IF (CylinderPosition>18) AND NOT CylinderExtractsLoadFromWarehouse AND NOT CylinderExtractsLoadFromWarehouseBlockHigh THEN
CylinderBehind:=TRUE; (*Il flag "CylinderBehind" e' attivo quando il cilindro sta tornardo indietro verso la posizione di riposo*)
END_IF;

(*generatore di vuoto*)
IF NOT VacuumGeneratorBlock THEN
	IF VacuumGenerator AND NOT ExpulsionAirVacuumVis THEN
		VacuumGeneratorSim:=TRUE; (*Simulo il funzionamento del generatore di vuoto solo se non è attivo anche il soffio di espulsione*)
		ELSE IF NOT VacuumGeneratorBlockHigh THEN
				VacuumGeneratorSim:=FALSE;
			END_IF;
	END_IF;
END_IF;

(*sensore di vuoto*)
IF VacuumGeneratorSim THEN
		IF NOT (VacuumGeneratorOkBlockHigh OR VacuumGeneratorOkBlockLow OR NOT ElementRotaryCharged) THEN
			VacuumGeneratorOk:=TRUE;
		END_IF;
	ELSE IF NOT (VacuumGeneratorOkBlockHigh OR VacuumGeneratorOkBlockLow OR NOT ElementRotaryCharged) THEN
				VacuumGeneratorOk:=FALSE;
		END_IF;
END_IF;

IF NOT ElementRotaryCharged THEN (*se non ho un pezzo sotto alla ventosa non si genera il vuoto*)
	VacuumGeneratorOk:=FALSE;
END_IF;

(*soffio di rilascio pezzo*)
IF NOT ExpulsionAirVacuumBlock THEN
	IF NOT VacuumGeneratorBlockHigh AND ExpulsionAirVacuum THEN (*se ho il pezzo sull'ascensore avvio il rilascio*)
		ExpulsionAirVacuumVis:=TRUE;
		ELSE IF NOT ExpulsionAirVacuumBlockHigh THEN
				ExpulsionAirVacuumVis:=FALSE;
			END_IF;
	END_IF;
END_IF;

(*sensore generazione di vuoto guasto: *)
IF VacuumGeneratorOkBlockHigh THEN
	VacuumGeneratorOk:=TRUE;
END_IF;
IF VacuumGeneratorOkBlockLow THEN
	VacuumGeneratorOk:=FALSE;
END_IF;

(*braccio rotante*)
IF NOT RotaryMakerVsVerificationBlock THEN
	IF (RotaryMakerVsVerification OR BlockedVsVerification)  AND RotaryPosition<=180 AND NOT BlockedVsWarehouse  THEN  (*Il braccio va verso la stazione di verifica quando non è già a fine corsa e il relativo comando e' attivo, oppure è bloccato alto*)
		RotaryPosition:=RotaryPosition+9;
		IF RotaryMakerVsVerificationBlockHigh THEN  (*simulo il bloccaggio del braccio in posizione di verifica*)
			BlockedVsVerification:=TRUE;
			ELSE BlockedVsVerification:=FALSE;
		END_IF;
	END_IF;
END_IF;

IF NOT RotaryMakerVsWarehouseBlock THEN
	IF (RotaryMakerVsWarehouse OR BlockedVsWarehouse) AND RotaryPosition>=0 AND NOT BlockedVsVerification THEN  (*Il braccio va verso il magazzino quando non è già a fine corsa e il relativo comando e' attivo, oppure è bloccato alto*)
		RotaryPosition:=RotaryPosition-9;
		IF RotaryMakerVsWarehouseBlockHigh THEN  (*simulo il bloccaggio del braccio in posizione magazzino*)
			BlockedVsWarehouse:=TRUE;
			ELSE BlockedVsWarehouse:=FALSE;
		END_IF;
	END_IF;
END_IF;

IF RotaryPosition<1 THEN  (*Il braccio giunge a fine corsa verso il magazzino ed il relativo sensore si attiva*)
	RotaryPosition:=0;
	IF NOT (RotaryMakerInPositionWarehouseBlockHigh OR RotaryMakerInPositionWarehouseBlockLow) THEN
		RotaryMakerInPositionWarehouse:=TRUE; (*Questo sensore e' attivo quando il cilindro e' in posizione retratta*)
	END_IF;
	ELSE IF NOT (RotaryMakerInPositionWarehouseBlockHigh OR RotaryMakerInPositionWarehouseBlockLow) THEN
			RotaryMakerInPositionWarehouse:=FALSE;
		END_IF;
END_IF;

(*sensore finecorsa inferiore braccio rotante guasto*)
IF RotaryMakerInPositionWarehouseBlockHigh THEN
	RotaryMakerInPositionWarehouse:=TRUE;
END_IF;
IF RotaryMakerInPositionWarehouseBlockLow THEN
	RotaryMakerInPositionWarehouse:=FALSE;
END_IF;

IF RotaryPosition>=180 THEN (*Il braccio giunge a fine corsa verso la verifica ed il relativo sensore si attiva*)
	RotaryPosition:=180;
	IF NOT (RotaryMakerInPositionVerificationBlockHigh OR RotaryMakerInPositionVerificationBlockLow) THEN
		RotaryMakerInPositionVerification:=TRUE; (*sensore*)
	END_IF;
	ELSE IF NOT (RotaryMakerInPositionVerificationBlockHigh OR RotaryMakerInPositionVerificationBlockLow) THEN
			RotaryMakerInPositionVerification:=FALSE;
		END_IF;
END_IF;

(*sensore finecorsa superiore braccio rotante guasto*)
IF RotaryMakerInPositionVerificationBlockHigh THEN
	RotaryMakerInPositionVerification:=TRUE;
END_IF;
IF RotaryMakerInPositionVerificationBlockLow THEN
	RotaryMakerInPositionVerification:=FALSE;
END_IF;

(*attivazione della fotocellula per l'interferenza braccioRotante-ascensore*)
IF NOT (VerificationBusyBlockHigh OR VerificationBusyBlockLow) THEN
	IF RotaryPosition>140  OR LiftPosition>10 THEN
		VerificationBusy:=TRUE;
		ELSE
			VerificationBusy:=FALSE;
	END_IF;
END_IF;

(*fotocellula interferenza guasta: *)
IF VerificationBusyBlockHigh THEN
	VerificationBusy:=TRUE;
END_IF;
IF VerificationBusyBlockLow THEN
	VerificationBusy:=FALSE;
END_IF;

(*Se gli elementi sono capovolti, nella simulazione grafica questo viene segnalato da una "O" scritta sul pezzo*)
IF ElementOneOverturned THEN
	ElementOneO:='O';
	ELSE  IF NOT ElementOneShort THEN
		ElementOneO:='' ;
	END_IF;
END_IF;

IF ElementTwoOverturned THEN
	ElementTwoO:='O';
	ELSE  IF NOT ElementTwoShort THEN
		ElementTwoO:='' ;
	END_IF;
END_IF;

IF ElementThreeOverturned THEN
	ElementThreeO:='O';
	ELSE  IF NOT ElementThreeShort THEN
		ElementThreeO:='' ;
	END_IF;
END_IF;

IF ElementFourOverturned THEN
	ElementFourO:='O';
	ELSE  IF NOT ElementFourShort THEN
		ElementFourO:='' ;
	END_IF;
END_IF;

IF ElementFiveOverturned THEN
	ElementFiveO:='O';
	ELSE  IF NOT ElementFiveShort THEN
		ElementFiveO:='' ;
	END_IF;
END_IF;

IF ElementSixOverturned THEN
	ElementSixO:='O';
	ELSE  IF NOT ElementSixShort THEN
		ElementSixO:='' ;
	END_IF;
END_IF;

IF ElementSevenOverturned THEN
	ElementSevenO:='O';
	ELSE  IF NOT ElementSevenShort THEN
		ElementSevenO:='' ;
	END_IF;
END_IF;

IF ElementEightOverturned THEN
	ElementEightO:='O';
	ELSE  IF NOT ElementEightShort THEN
		ElementEightO:='' ;
	END_IF;
END_IF;

IF ElementWaitingOverturned THEN
	ElementWaitingO:='O';
	ELSE  IF NOT ElementWaitingShort THEN
		ElementWaitingO:='' ;
	END_IF;
END_IF;

IF ElementRotaryOverturned THEN
	ElementRotaryO:='O';
	ELSE  IF NOT ElementRotaryShort THEN
		ElementRotaryO:='' ;
	END_IF;
END_IF;

IF ElementVerificationOverturned THEN
	ElementVerificationO:='O';
	ELSE  IF NOT ElementVerificationShort THEN
		ElementVerificationO:='' ;
	END_IF;
END_IF;

IF ElementMeasureOverturned THEN
	ElementMeasureO:='O';
	ELSE  IF NOT ElementMeasureShort THEN
		ElementMeasureO:='' ;
	END_IF;
END_IF;

IF ElementAirOverturned THEN (*se c'era un pezzo corto ora è già stato scartato quindi nn lo considero più*)
	ElementAirO:='O'; ELSE
	ElementAirO:='' ;
END_IF;

IF ElementOneTableOverturned THEN
	ElementOneTableO:='O'; ELSE
	ElementOneTableO:='' ;
END_IF;

(*Se gli elementi sono corti, nella simulazione grafica questo viene segnalato da una "S" scritta sul pezzo*)
IF ElementOneShort THEN
	ElementOneO:='S';
	ELSE IF NOT ElementOneOverturned THEN
		ElementOneO:='' ;
	END_IF;
END_IF;

IF ElementTwoShort THEN
	ElementTwoO:='S';
	ELSE IF NOT ElementTwoOverturned THEN
		ElementTwoO:='' ;
	END_IF;
END_IF;

IF ElementThreeShort THEN
	ElementThreeO:='S';
	ELSE IF NOT ElementThreeOverturned THEN
		ElementThreeO:='' ;
	END_IF;
END_IF;

IF ElementFourShort THEN
	ElementFourO:='S';
	ELSE IF NOT ElementFourOverturned THEN
		ElementFourO:='' ;
	END_IF;
END_IF;

IF ElementFiveShort THEN
	ElementFiveO:='S';
	ELSE IF NOT ElementFiveOverturned THEN
		ElementFiveO:='' ;
	END_IF;
END_IF;

IF ElementSixShort THEN
	ElementSixO:='S';
	ELSE IF NOT ElementSixOverturned THEN
		ElementSixO:='' ;
	END_IF;
END_IF;

IF ElementSevenShort THEN
	ElementSevenO:='S';
	ELSE IF NOT ElementSevenOverturned THEN
		ElementSevenO:='' ;
	END_IF;
END_IF;

IF ElementEightShort THEN
	ElementEightO:='S';
	ELSE IF NOT ElementEightOverturned THEN
		ElementEightO:='' ;
	END_IF;
END_IF;

IF ElementWaitingShort THEN
	ElementWaitingO:='S';
	ELSE IF NOT ElementWaitingOverturned THEN
		ElementWaitingO:='' ;
	END_IF;
END_IF;


IF ElementRotaryShort THEN
	ElementRotaryO:='S';
	ELSE IF NOT ElementRotaryOverturned THEN
		ElementRotaryO:='' ;
	END_IF;
END_IF;

IF ElementVerificationShort THEN
	ElementVerificationO:='S';
	ELSE IF NOT ElementVerificationOverturned THEN
		ElementVerificationO:='' ;
	END_IF;
END_IF;

IF ElementMeasureShort THEN
	ElementMeasureO:='S';
	ELSE IF NOT ElementMeasureOverturned THEN
		ElementMeasureO:='' ;
	END_IF;
END_IF;
END_PROGRAM

(* POU 0_Simulation/PlantVerification, ST *)
PROGRAM PlantVerification
VAR
	NoElement: BOOL; (*variabile che segnala se il pezzo è gia stato preso dal rotary maker (necessaria nel caso di estrattore-basi bloccato alto) *)
	BlockedHigh: BOOL; (*flag che segnala il bloccaggio alto dell'ascensore*)
	BlockedLow: BOOL; (*flag che segnala il bloccaggio basso dell'ascensore*)
END_VAR
(* Valore iniziale braccio rotante*)
IF FLAGRotaryPosition
THEN 	FLAGRotaryPosition:=FALSE;
		RotaryPosition:=RotaryPositionInitialVis+RotaryPosition;
END_IF;

(* Valore iniziale ascensore*)
IF FLAGLiftPosition
THEN 	FLAGLiftPosition:=FALSE;
		LiftPosition:=LiftPositionInitialVis+LiftPosition;
END_IF;

(*elemento in attesa di essere caricato dal RotaryMaker*)
IF CylinderExtractionLoadInExtensivePosition AND ElementOneCharged AND NOT CylinderExtractionLoadInExtensivePositionBlockHigh THEN	(*Quando il cilindro di espulsione dal magazzino e' arrivato a fine corsa, viene reso visibile il pezzo in posizione di attesa*)
	ElementWaitingCharged:=TRUE;
	ElementWaitingRed:=ElementOneRed;
	ElementWaitingBlack:=ElementOneBlack;
	ElementWaitingSilver:=ElementOneSilver;
	ElementWaitingOverturned:=ElementOneOverturned;
	ElementWaitingShort:=ElementOneShort;
	ElementOneCharged:=FALSE;
	NoElement:=TRUE;
END_IF;

IF CylinderBehind THEN
	NoElement:=FALSE;
END_IF;

(*elemento caricato dal braccio rotante*)
IF ElementWaitingCharged  AND RotaryMakerInPositionWarehouse THEN
	ElementRotaryCharged:=TRUE;
	ElementRotaryRed:=ElementWaitingRed;
	ElementRotaryBlack:=ElementWaitingBlack;
	ElementRotarySilver:=ElementWaitingSilver;
	ElementRotaryOverturned:=ElementWaitingOverturned;
	ElementRotaryShort:=ElementWaitingShort;
	ElementWaitingCharged:=FALSE;
END_IF;

(*----------------Plant della stazione di verifica---------------*)
(*ascensore*)
IF NOT  ToLiftCylinderToMeasureLoadBlock THEN
	IF (ToLiftCylinderToMeasureLoad OR BlockedHigh) AND LiftPosition<=140 AND NOT BlockedLow THEN (*l'ascensore sale quando Il relativo comando e' attivo o è bloccato alto*)
		LiftPosition:=LiftPosition+7;
		IF ToLiftCylinderToMeasureLoadBlockHigh THEN  (*simulo il bloccaggio dell'ascensore in alto*)
			BlockedHigh:=TRUE;
			ELSE BlockedHigh:=FALSE;
		END_IF;
	END_IF;
END_IF;

IF NOT  ToLowerCylinderToMeasureLoadBlock THEN
	IF (ToLowerCylinderToMeasureLoad OR BlockedLow) AND LiftPosition>=0 AND NOT BlockedHigh THEN (*l'ascensore scende quando Il relativo comando e' attivo o è bloccato alto*)
		LiftPosition:=LiftPosition-7;
		IF ToLowerCylinderToMeasureLoadBlockHigh THEN  (*simulo il bloccaggio dell'ascensore in basso*)
			BlockedLow:=TRUE;
			ELSE BlockedLow:=FALSE;
		END_IF;
	END_IF;
END_IF;

IF LiftPosition<1 THEN
	LiftPosition:=0;
END_IF;

IF LiftPosition>=140 THEN
	LiftPosition:=140;
END_IF;

(*sensore di finecorsa inferiore ascensore*)
IF NOT (CylinderDownToMeasureLoadBlockHigh OR CylinderDownToMeasureLoadBlockLow) THEN
	IF (LiftPosition>=0 AND LiftPosition<=15) OR (LiftPosition>=30 AND LiftPosition<=45) THEN   (*Sensore di finecorsa inferiore dell'ascensore*)
			CylinderDownToMeasureLoad:=TRUE;
		ELSE CylinderDownToMeasureLoad:=FALSE;
	END_IF;
END_IF;

(*sensore di finecorsa inferiore ascensore guasto*)
IF CylinderDownToMeasureLoadBlockHigh THEN
	CylinderDownToMeasureLoad:=TRUE;
END_IF;
IF CylinderDownToMeasureLoadBlockLow THEN
	CylinderDownToMeasureLoad:=FALSE;
END_IF;

(*sensore di finecorsa superiore ascensore*)
IF NOT (CylinderUpToMeasureLoadBlockHigh OR CylinderUpToMeasureLoadBlockLow) THEN
	IF LiftPosition=140 THEN
			CylinderUpToMeasureLoad:=TRUE;
		ELSE CylinderUpToMeasureLoad:=FALSE;
	END_IF;
END_IF;

(*sensore di finecorsa superiore ascensore guasto*)
IF CylinderUpToMeasureLoadBlockHigh THEN
	CylinderUpToMeasureLoad:=TRUE;
END_IF;
IF CylinderUpToMeasureLoadBlockLow THEN
	CylinderUpToMeasureLoad:=FALSE;
END_IF;

(*cilindro di espulsione sull'ascensore*)
IF NOT ToExtendCylinderOfExtractionVsGuideBlock THEN
	IF ToExtendCylinderOfExtractionVsGuide AND CylinderOfExtractionPosition<=80 THEN  (*Quando il relativo comando e' attivo, il cilindro di espulsione sull'ascensore e' attivo, altrimenti torna a fine corsa*)
			CylinderOfExtractionPosition:=CylinderOfExtractionPosition+4;
		ELSE IF (NOT ToExtendCylinderOfExtractionVsGuide  AND CylinderOfExtractionPosition>=0  OR Fault) AND NOT ToExtendCylinderOfExtractionVsGuideBlockHigh THEN
				CylinderOfExtractionPosition:=CylinderOfExtractionPosition-4;
			END_IF;
	END_IF;
END_IF;

(*sensore di finecorsa cilindro di espulsione (solo inferiore) *)
IF CylinderOfExtractionPosition<1 THEN	(*Simulazione del cilindro di espulsione scarti*)
	CylinderOfExtractionPosition:=0;
	IF NOT (CylinderOfExtractionInRetroactivePositionBlockHigh OR CylinderOfExtractionInRetroactivePositionBlockLow) THEN
		CylinderOfExtractionInRetroactivePosition:=TRUE;
	END_IF;
	ELSE IF NOT (CylinderOfExtractionInRetroactivePositionBlockHigh OR CylinderOfExtractionInRetroactivePositionBlockLow) THEN
			CylinderOfExtractionInRetroactivePosition:=FALSE;
		END_IF;
END_IF;

(*sensore di finecorsa cilindro di espulsione (solo inferiore) guasto *)
IF CylinderOfExtractionInRetroactivePositionBlockHigh THEN
	CylinderOfExtractionInRetroactivePosition:=TRUE;
END_IF;
IF CylinderOfExtractionInRetroactivePositionBlockLow THEN
	CylinderOfExtractionInRetroactivePosition:=FALSE;
END_IF;

IF CylinderOfExtractionPosition>=80 THEN
	CylinderOfExtractionPosition:=80;
END_IF;

IF CylinderOfExtractionPosition>=75 THEN
	ElementVerificationCharged:=FALSE; (*Se ho espulso il pezzo non ho più l'elemento in verifica*)
END_IF;

(*verifica colore*)
IF NOT (ColourMeasurementBlockHigh OR ColourMeasurementBlockLow) THEN
	IF ElementVerificationBlack  AND CylinderOfExtractionPosition=0 THEN	(*Se l'elemento e' nero, il sensore di rilevamento colore non si accende*)
		ColourMeasurement:=FALSE;
	END_IF;
	IF (ElementVerificationSilver OR ElementVerificationRed)  AND CylinderOfExtractionPosition<70 AND (ElementVerificationCharged OR ElementMeasureCharged) THEN
			ColourMeasurement:=TRUE;
		ELSE ColourMeasurement:=FALSE;
	END_IF;
END_IF;

(*sensore di verifica colore guasto*)
IF ColourMeasurementBlockHigh THEN
	ColourMeasurement:=TRUE;
END_IF;
IF ColourMeasurementBlockLow THEN
	ColourMeasurement:=FALSE;
END_IF;

IF MisuratorPosition>=40 THEN
	MisuratorPosition:=40;
END_IF;

IF MisuratorPosition<1 THEN
	MisuratorPosition:=0;
END_IF;

IF (LiftPosition>135 AND MisuratorPosition>=0 AND (ElementVerificationCharged OR ElementMeasureCharged)) AND CylinderOfExtractionPosition<50  THEN
			MisuratorPosition:=MisuratorPosition-12;
END_IF;

(*uscita misuratore*)
IF NOT (MeasurementNotOkBlockHigh OR MeasurementNotOkBlockLow) THEN
	IF ElementMeasureBlack THEN	(*Se l'elemento è nero (cioè basso), la misura dà in uscita FALSE*)
		MeasurementNotOk:=FALSE;
	END_IF;
	IF (ElementMeasureSilver OR ElementMeasureRed) AND NOT ElementMeasureShort AND CylinderOfExtractionPosition<70 AND ElementMeasureCharged THEN (*Se l'elemento è chiaro normale (cioè alto), la misura dà in uscita TRUE*)
				MeasurementNotOk:=TRUE;
			ELSE MeasurementNotOk:=FALSE;
		END_IF;
	IF ElementMeasureShort THEN (*Se l'elemento è chiaro corto, la misura dà in uscita FALSE*)
		MeasurementNotOk:=FALSE;
		IF LiftPosition>2 THEN
				ElementVerificationCharged:=TRUE;  (*rivisualizzo l'elemento corto in Verification e lo nascondo da Measure*)
				ElementMeasureCharged:=FALSE;
				ElementVerificationShort:=ElementMeasureShort;
		END_IF;
	END_IF;
END_IF;

IF NOT ElementVerificationCharged THEN  (*se ho espulso il pezzo corto resetto le variabili che lo identificavano*)
		ElementVerificationShort:=FALSE;
		ElementMeasureShort:=FALSE;
END_IF;

(*sensore di misura rotto*)
IF MeasurementNotOkBlockHigh THEN
	MeasurementNotOk:=TRUE;
END_IF;
IF MeasurementNotOkBlockLow THEN
	MeasurementNotOk:=FALSE;
END_IF;

(*elemento nella stazione di  verifica*)
IF RotaryMakerInPositionVerification AND ElementRotaryCharged AND NOT VacuumGeneratorBlockHigh THEN	(*Quando il braccio e' in posizione di verifica, l'elemento in questa posizione diventa visibile*)
	ElementVerificationCharged:=TRUE;
	ElementVerificationRed:=ElementRotaryRed;
	ElementVerificationBlack:=ElementRotaryBlack;
	ElementVerificationSilver:=ElementRotarySilver;
	ElementVerificationOverturned:=ElementRotaryOverturned;
	ElementVerificationShort:=ElementRotaryShort;
	ElementRotaryCharged:=FALSE;
	ReadyForRotaryMaker:=FALSE;
END_IF;

